SPLINE
SPL {X  -157.513, Y  +354.453, Z    +0.000, E1  +340.941, E3 -376360.122}
SPL {X  -159.408, Y  +368.861, Z    +0.000, E1  +348.865, E3 -376369.545}
SPL {X  -159.941, Y  +378.532, Z    +0.000, E1  +354.551, E3 -376373.150}
SPL {X  -159.990, Y  +383.966, Z    +0.000, E1  +358.149, E3 -376374.602}
SPL {X  -159.990, Y  +388.001, Z    +0.000, E1  +361.086, E3 -376375.537}
SPL {X  -159.990, Y  +392.647, Z    +0.000, E1  +364.974, E3 -376376.676}
SPL {X  -159.990, Y  +397.943, Z    +0.000, E1  +369.963, E3 -376378.260}
SPL {X  -159.990, Y  +406.530, Z    +0.000, E1  +377.917, E3 -376382.158}
SPL {X  -159.990, Y  +429.014, Z    +0.000, E1  +392.438, E3 -376400.815}
SPL {X  -159.990, Y  +437.635, Z    +0.000, E1  +395.495, E3 -376411.047}
SPL {X  -159.990, Y  +460.330, Z    +0.000, E1  +398.908, E3 -376451.734}
SPL {X  -159.990, Y  +464.953, Z    +0.000, E1  +398.907, E3 -376463.893}
SPL {X  -159.990, Y  +469.353, Z    +0.000, E1  +398.902, E3 -376475.473}
SPL {X  -159.990, Y  +475.034, Z    +0.000, E1  +398.936, E3 -376490.388}
SPL {X  -159.990, Y  +481.308, Z    +0.000, E1  +398.917, E3 -376506.899}
SPL {X  -159.990, Y  +486.996, Z    +0.000, E1  +398.928, E3 -376521.806}
SPL {X  -159.990, Y  +492.629, Z    +0.000, E1  +398.922, E3 -376536.613}
SPL {X  -159.990, Y  +497.431, Z    +0.000, E1  +398.905, E3 -376549.279}
SPL {X  -159.990, Y  +502.093, Z    +0.000, E1  +398.909, E3 -376561.554}
SPL {X  -159.990, Y  +507.821, Z    +0.000, E1  +398.930, E3 -376576.574}
SPL {X  -159.990, Y  +513.533, Z    +0.000, E1  +398.910, E3 -376591.633}
SPL {X  -159.990, Y  +518.435, Z    +0.000, E1  +398.905, E3 -376604.529}
SPL {X  -159.990, Y  +523.478, Z    +0.000, E1  +398.918, E3 -376617.757}
SPL {X  -159.990, Y  +528.627, Z    +0.000, E1  +398.910, E3 -376631.311}
SPL {X  -159.990, Y  +534.392, Z    +0.000, E1  +398.932, E3 -376646.441}
SPL {X  -159.990, Y  +540.299, Z    +0.000, E1  +398.912, E3 -376662.015}
SPL {X  -159.990, Y  +545.676, Z    +0.000, E1  +398.913, E3 -376676.153}
SPL {X  -159.990, Y  +550.777, Z    +0.000, E1  +398.906, E3 -376689.572}
SPL {X  -159.990, Y  +556.271, Z    +0.000, E1  +398.927, E3 -376703.975}
SPL {X  -159.990, Y  +561.696, Z    +0.000, E1  +398.912, E3 -376718.244}
SPL {X  -159.990, Y  +566.650, Z    +0.000, E1  +398.917, E3 -376731.258}
SPL {X  -159.990, Y  +571.814, Z    +0.000, E1  +398.914, E3 -376744.861}
SPL {X  -159.990, Y  +577.636, Z    +0.000, E1  +398.929, E3 -376760.158}
SPL {X  -159.990, Y  +583.167, Z    +0.000, E1  +398.906, E3 -376774.734}
SPL {X  -159.990, Y  +587.761, Z    +0.000, E1  +398.902, E3 -376786.819}
SPL {X  -159.990, Y  +592.962, Z    +0.000, E1  +398.925, E3 -376800.463}
SPL {X  -159.990, Y  +597.767, Z    +0.000, E1  +398.897, E3 -376813.138}
SPL {X  -159.990, Y  +602.727, Z    +0.000, E1  +398.920, E3 -376826.149}
SPL {X  -159.990, Y  +608.112, Z    +0.000, E1  +398.911, E3 -376840.323}
SPL {X  -159.990, Y  +613.039, Z    +0.000, E1  +398.906, E3 -376853.286}
SPL {X  -159.990, Y  +618.087, Z    +0.000, E1  +398.915, E3 -376866.544}
SPL {X  -159.990, Y  +623.264, Z    +0.000, E1  +398.906, E3 -376880.179}
SPL {X  -159.990, Y  +628.669, Z    +0.000, E1  +398.928, E3 -376894.347}
SPL {X  -159.990, Y  +634.089, Z    +0.000, E1  +398.907, E3 -376908.623}
SPL {X  -159.990, Y  +638.639, Z    +0.000, E1  +398.904, E3 -376920.608}
SPL {X  -159.990, Y  +643.555, Z    +0.000, E1  +398.910, E3 -376933.528}
SPL {X  -159.990, Y  +649.380, Z    +0.000, E1  +398.930, E3 -376948.806}
SPL {X  -159.990, Y  +654.813, Z    +0.000, E1  +398.905, E3 -376963.131}
SPL {X  -159.990, Y  +660.353, Z    +0.000, E1  +398.930, E3 -376977.662}
SPL {X  -159.990, Y  +665.703, Z    +0.000, E1  +398.903, E3 -376991.769}
SPL {X  -159.990, Y  +669.966, Z    +0.000, E1  +398.902, E3 -377002.976}
SPL {X  -159.954, Y  +674.895, Z    +0.000, E1  +398.910, E3 -377015.956}
SPL {X  -159.761, Y  +680.061, Z    +0.000, E1  +398.873, E3 -377029.735}
SPL {X  -159.443, Y  +684.716, Z    +0.000, E1  +398.815, E3 -377042.300}
SPL {X  -158.962, Y  +689.604, Z    +0.000, E1  +398.740, E3 -377055.669}
SPL {X  -158.318, Y  +694.567, Z    +0.000, E1  +398.614, E3 -377069.430}
SPL {X  -157.472, Y  +699.775, Z    +0.000, E1  +398.483, E3 -377083.990}
SPL {X  -156.506, Y  +704.705, Z    +0.000, E1  +398.294, E3 -377097.990}
SPL {X  -155.357, Y  +709.721, Z    +0.000, E1  +398.108, E3 -377112.345}
SPL {X  -154.005, Y  +714.851, Z    +0.000, E1  +397.854, E3 -377127.240}
SPL {X  -153.100, Y  +717.944, Z    +0.000, E1  +397.652, E3 -377136.350}
SPL {X  -151.080, Y  +724.146, Z    +0.000, E1  +393.201, E3 -377192.396}
ENDSPLINE

SPLINE
SPL {X  -157.921, Y  +697.149, Z    +0.000, E1  +377.701, E3 -377243.957}
SPL {X  -159.579, Y  +682.959, Z    +0.000, E1  +369.793, E3 -377251.905}
SPL {X  -159.938, Y  +675.561, Z    +0.000, E1  +365.399, E3 -377254.327}
SPL {X  -159.990, Y  +669.910, Z    +0.000, E1  +361.710, E3 -377255.618}
SPL {X  -159.990, Y  +665.465, Z    +0.000, E1  +358.378, E3 -377256.535}
SPL {X  -159.990, Y  +661.791, Z    +0.000, E1  +355.213, E3 -377257.373}
SPL {X  -159.990, Y  +656.991, Z    +0.000, E1  +350.742, E3 -377258.792}
SPL {X  -159.990, Y  +648.067, Z    +0.000, E1  +342.328, E3 -377262.522}
SPL {X  -159.990, Y  +620.451, Z    +0.000, E1  +325.419, E3 -377286.369}
SPL {X  -159.990, Y  +591.256, Z    +0.000, E1  +319.966, E3 -377332.863}
SPL {X  -159.990, Y  +586.740, Z    +0.000, E1  +319.956, E3 -377344.253}
SPL {X  -159.990, Y  +581.814, Z    +0.000, E1  +319.956, E3 -377356.692}
SPL {X  -159.990, Y  +577.274, Z    +0.000, E1  +319.964, E3 -377368.170}
SPL {X  -159.990, Y  +572.933, Z    +0.000, E1  +319.959, E3 -377379.111}
SPL {X  -159.990, Y  +568.504, Z    +0.000, E1  +319.956, E3 -377390.274}
SPL {X  -159.990, Y  +564.427, Z    +0.000, E1  +319.959, E3 -377400.560}
SPL {X  -159.990, Y  +558.823, Z    +0.000, E1  +319.916, E3 -377414.639}
SPL {X  -159.990, Y  +553.571, Z    +0.000, E1  +319.954, E3 -377427.921}
SPL {X  -159.990, Y  +549.413, Z    +0.000, E1  +319.938, E3 -377438.387}
SPL {X  -159.990, Y  +543.439, Z    +0.000, E1  +319.921, E3 -377453.475}
SPL {X  -159.990, Y  +537.213, Z    +0.000, E1  +319.937, E3 -377469.217}
SPL {X  -159.990, Y  +530.667, Z    +0.000, E1  +319.910, E3 -377485.675}
SPL {X  -159.990, Y  +523.984, Z    +0.000, E1  +319.922, E3 -377502.542}
SPL {X  -159.990, Y  +496.806, Z    +0.000, E1  +312.216, E3 -377516.457}
SPL {X  -159.990, Y  +490.245, Z    +0.000, E1  +312.831, E3 -377532.988}
SPL {X  -159.990, Y  +484.831, Z    +0.000, E1  +314.066, E3 -377551.220}
SPL {X  -159.990, Y  +480.580, Z    +0.000, E1  +315.242, E3 -377566.907}
SPL {X  -159.990, Y  +476.546, Z    +0.000, E1  +316.165, E3 -377581.202}
SPL {X  -159.990, Y  +472.671, Z    +0.000, E1  +317.192, E3 -377596.029}
SPL {X  -159.990, Y  +468.809, Z    +0.000, E1  +318.343, E3 -377611.957}
SPL {X  -159.990, Y  +465.057, Z    +0.000, E1  +319.375, E3 -377627.116}
SPL {X  -159.990, Y  +461.409, Z    +0.000, E1  +319.848, E3 -377639.015}
SPL {X  -159.990, Y  +456.934, Z    +0.000, E1  +319.854, E3 -377650.291}
SPL {X  -159.990, Y  +452.940, Z    +0.000, E1  +319.854, E3 -377660.336}
SPL {X  -159.990, Y  +448.856, Z    +0.000, E1  +319.859, E3 -377670.619}
SPL {X  -159.990, Y  +443.741, Z    +0.000, E1  +319.827, E3 -377683.437}
SPL {X  -159.990, Y  +436.703, Z    +0.000, E1  +319.809, E3 -377701.119}
SPL {X  -159.990, Y  +430.690, Z    +0.000, E1  +319.854, E3 -377716.312}
SPL {X  -159.990, Y  +426.145, Z    +0.000, E1  +319.853, E3 -377727.752}
SPL {X  -159.990, Y  +421.880, Z    +0.000, E1  +319.860, E3 -377738.485}
SPL {X  -159.990, Y  +417.572, Z    +0.000, E1  +319.852, E3 -377749.311}
SPL {X  -159.990, Y  +412.619, Z    +0.000, E1  +319.850, E3 -377761.803}
SPL {X  -159.990, Y  +406.264, Z    +0.000, E1  +319.825, E3 -377777.751}
SPL {X  -159.990, Y  +400.535, Z    +0.000, E1  +319.859, E3 -377792.214}
SPL {X  -159.990, Y  +396.024, Z    +0.000, E1  +319.860, E3 -377803.570}
SPL {X  -159.990, Y  +391.614, Z    +0.000, E1  +319.860, E3 -377814.663}
SPL {X  -159.990, Y  +387.212, Z    +0.000, E1  +319.859, E3 -377825.736}
SPL {X  -159.990, Y  +382.743, Z    +0.000, E1  +319.857, E3 -377836.977}
SPL {X  -159.925, Y  +377.946, Z    +0.000, E1  +319.864, E3 -377849.114}
SPL {X  -159.703, Y  +372.915, Z    +0.000, E1  +319.904, E3 -377862.014}
SPL {X  -159.358, Y  +368.290, Z    +0.000, E1  +319.961, E3 -377873.976}
SPL {X  -158.955, Y  +364.333, Z    +0.000, E1  +320.046, E3 -377884.379}
SPL {X  -158.482, Y  +360.589, Z    +0.000, E1  +320.125, E3 -377894.305}
SPL {X  -157.729, Y  +355.695, Z    +0.000, E1  +320.237, E3 -377907.378}
SPL {X  -156.893, Y  +351.173, Z    +0.000, E1  +320.410, E3 -377919.661}
SPL {X  -156.148, Y  +347.650, Z    +0.000, E1  +320.549, E3 -377929.307}
SPL {X  -155.268, Y  +343.918, Z    +0.000, E1  +320.696, E3 -377939.588}
SPL {X  -153.936, Y  +338.906, Z    +0.000, E1  +320.911, E3 -377953.527}
SPL {X  -152.628, Y  +334.526, Z    +0.000, E1  +321.188, E3 -377965.929}
SPL {X  -151.010, Y  +329.654, Z    +0.000, E1  +326.674, E3 -378023.765}
ENDSPLINE

SPLINE
SPL {X  -157.513, Y  +354.453, Z    +0.000, E1  +340.941, E3 -378069.799}
SPL {X  -159.408, Y  +368.861, Z    +0.000, E1  +348.865, E3 -378079.222}
SPL {X  -159.941, Y  +378.532, Z    +0.000, E1  +354.551, E3 -378082.828}
SPL {X  -159.990, Y  +383.966, Z    +0.000, E1  +358.149, E3 -378084.280}
SPL {X  -159.990, Y  +388.001, Z    +0.000, E1  +361.086, E3 -378085.215}
SPL {X  -159.990, Y  +392.647, Z    +0.000, E1  +364.974, E3 -378086.353}
SPL {X  -159.990, Y  +397.943, Z    +0.000, E1  +369.963, E3 -378087.938}
SPL {X  -159.990, Y  +407.689, Z    +0.000, E1  +378.860, E3 -378092.592}
SPL {X  -159.990, Y  +434.822, Z    +0.000, E1  +394.625, E3 -378117.136}
SPL {X  -159.990, Y  +460.330, Z    +0.000, E1  +398.908, E3 -378161.412}
SPL {X  -159.990, Y  +464.953, Z    +0.000, E1  +398.907, E3 -378173.570}
SPL {X  -159.990, Y  +469.353, Z    +0.000, E1  +398.902, E3 -378185.150}
SPL {X  -159.990, Y  +475.034, Z    +0.000, E1  +398.936, E3 -378200.065}
SPL {X  -159.990, Y  +481.308, Z    +0.000, E1  +398.917, E3 -378216.576}
SPL {X  -159.990, Y  +485.396, Z    +0.000, E1  +398.893, E3 -378227.336}
SPL {X  -159.990, Y  +489.893, Z    +0.000, E1  +398.930, E3 -378239.091}
SPL {X  -159.990, Y  +496.271, Z    +0.000, E1  +398.942, E3 -378255.847}
SPL {X  -159.990, Y  +502.093, Z    +0.000, E1  +398.909, E3 -378271.231}
SPL {X  -159.990, Y  +507.821, Z    +0.000, E1  +398.930, E3 -378286.251}
SPL {X  -159.990, Y  +513.533, Z    +0.000, E1  +398.910, E3 -378301.311}
SPL {X  -159.990, Y  +518.435, Z    +0.000, E1  +398.905, E3 -378314.206}
SPL {X  -159.990, Y  +523.478, Z    +0.000, E1  +398.918, E3 -378327.435}
SPL {X  -159.990, Y  +528.627, Z    +0.000, E1  +398.910, E3 -378340.988}
SPL {X  -159.990, Y  +533.053, Z    +0.000, E1  +398.899, E3 -378352.646}
SPL {X  -159.990, Y  +537.174, Z    +0.000, E1  +398.910, E3 -378363.460}
SPL {X  -159.990, Y  +541.259, Z    +0.000, E1  +398.888, E3 -378374.260}
SPL {X  -159.990, Y  +545.676, Z    +0.000, E1  +398.913, E3 -378385.831}
SPL {X  -159.990, Y  +550.777, Z    +0.000, E1  +398.906, E3 -378399.250}
SPL {X  -159.990, Y  +554.638, Z    +0.000, E1  +398.890, E3 -378409.420}
SPL {X  -159.990, Y  +557.678, Z    +0.000, E1  +398.893, E3 -378417.396}
SPL {X  -159.990, Y  +561.696, Z    +0.000, E1  +398.912, E3 -378427.922}
SPL {X  -159.990, Y  +566.650, Z    +0.000, E1  +398.917, E3 -378440.935}
SPL {X  -159.990, Y  +571.814, Z    +0.000, E1  +398.914, E3 -378454.538}
SPL {X  -159.990, Y  +576.364, Z    +0.000, E1  +398.896, E3 -378466.541}
SPL {X  -159.990, Y  +582.060, Z    +0.000, E1  +398.942, E3 -378481.447}
SPL {X  -159.990, Y  +589.106, Z    +0.000, E1  +398.939, E3 -378499.978}
SPL {X  -159.990, Y  +596.185, Z    +0.000, E1  +398.945, E3 -378518.587}
SPL {X  -159.990, Y  +602.727, Z    +0.000, E1  +398.920, E3 -378535.826}
SPL {X  -159.990, Y  +608.112, Z    +0.000, E1  +398.911, E3 -378550.001}
SPL {X  -159.990, Y  +614.125, Z    +0.000, E1  +398.936, E3 -378565.776}
SPL {X  -159.990, Y  +619.061, Z    +0.000, E1  +398.894, E3 -378578.807}
SPL {X  -159.990, Y  +623.264, Z    +0.000, E1  +398.906, E3 -378589.856}
SPL {X  -159.990, Y  +628.669, Z    +0.000, E1  +398.928, E3 -378604.025}
SPL {X  -159.990, Y  +634.089, Z    +0.000, E1  +398.907, E3 -378618.300}
SPL {X  -159.990, Y  +638.639, Z    +0.000, E1  +398.904, E3 -378630.286}
SPL {X  -159.990, Y  +644.750, Z    +0.000, E1  +398.946, E3 -378646.291}
SPL {X  -159.990, Y  +650.458, Z    +0.000, E1  +398.900, E3 -378661.364}
SPL {X  -159.990, Y  +654.813, Z    +0.000, E1  +398.905, E3 -378672.808}
SPL {X  -159.990, Y  +660.353, Z    +0.000, E1  +398.930, E3 -378687.339}
SPL {X  -159.990, Y  +665.703, Z    +0.000, E1  +398.903, E3 -378701.447}
SPL {X  -159.990, Y  +669.966, Z    +0.000, E1  +398.902, E3 -378712.653}
SPL {X  -159.954, Y  +674.895, Z    +0.000, E1  +398.910, E3 -378725.633}
SPL {X  -159.761, Y  +680.061, Z    +0.000, E1  +398.873, E3 -378739.412}
SPL {X  -159.443, Y  +684.716, Z    +0.000, E1  +398.815, E3 -378751.977}
SPL {X  -158.962, Y  +689.604, Z    +0.000, E1  +398.740, E3 -378765.346}
SPL {X  -158.139, Y  +695.766, Z    +0.000, E1  +398.623, E3 -378782.392}
SPL {X  -157.275, Y  +700.848, Z    +0.000, E1  +398.415, E3 -378796.744}
SPL {X  -156.506, Y  +704.705, Z    +0.000, E1  +398.294, E3 -378807.668}
SPL {X  -155.357, Y  +709.721, Z    +0.000, E1  +398.108, E3 -378822.023}
SPL {X  -154.286, Y  +713.838, Z    +0.000, E1  +397.877, E3 -378834.005}
SPL {X  -153.345, Y  +717.131, Z    +0.000, E1  +397.713, E3 -378843.619}
SPL {X  -151.080, Y  +724.146, Z    +0.000, E1  +393.201, E3 -378902.073}
ENDSPLINE

SPLINE
SPL {X  -157.921, Y  +697.149, Z    +0.000, E1  +377.701, E3 -378953.634}
SPL {X  -159.579, Y  +682.959, Z    +0.000, E1  +369.793, E3 -378961.582}
SPL {X  -159.938, Y  +675.561, Z    +0.000, E1  +365.399, E3 -378964.005}
SPL {X  -159.990, Y  +669.910, Z    +0.000, E1  +361.710, E3 -378965.295}
SPL {X  -159.990, Y  +665.465, Z    +0.000, E1  +358.378, E3 -378966.213}
SPL {X  -159.990, Y  +661.791, Z    +0.000, E1  +355.213, E3 -378967.051}
SPL {X  -159.990, Y  +656.991, Z    +0.000, E1  +350.742, E3 -378968.470}
SPL {X  -159.990, Y  +648.067, Z    +0.000, E1  +342.328, E3 -378972.199}
SPL {X  -159.990, Y  +620.451, Z    +0.000, E1  +325.419, E3 -378996.047}
SPL {X  -159.990, Y  +591.256, Z    +0.000, E1  +319.966, E3 -379042.540}
SPL {X  -159.990, Y  +586.740, Z    +0.000, E1  +319.956, E3 -379053.930}
SPL {X  -159.990, Y  +581.814, Z    +0.000, E1  +319.956, E3 -379066.370}
SPL {X  -159.990, Y  +577.274, Z    +0.000, E1  +319.964, E3 -379077.847}
SPL {X  -159.990, Y  +572.933, Z    +0.000, E1  +319.959, E3 -379088.789}
SPL {X  -159.990, Y  +568.504, Z    +0.000, E1  +319.956, E3 -379099.951}
SPL {X  -159.990, Y  +563.189, Z    +0.000, E1  +319.932, E3 -379113.325}
SPL {X  -159.990, Y  +557.707, Z    +0.000, E1  +319.949, E3 -379127.180}
SPL {X  -159.990, Y  +552.104, Z    +0.000, E1  +319.922, E3 -379141.255}
SPL {X  -159.990, Y  +545.912, Z    +0.000, E1  +319.929, E3 -379156.904}
SPL {X  -159.990, Y  +540.054, Z    +0.000, E1  +319.939, E3 -379171.732}
SPL {X  -159.990, Y  +535.835, Z    +0.000, E1  +319.966, E3 -379182.412}
SPL {X  -159.990, Y  +530.667, Z    +0.000, E1  +319.910, E3 -379195.353}
SPL {X  -159.990, Y  +523.984, Z    +0.000, E1  +319.922, E3 -379212.219}
SPL {X  -159.990, Y  +496.806, Z    +0.000, E1  +312.216, E3 -379226.134}
SPL {X  -159.990, Y  +490.245, Z    +0.000, E1  +312.831, E3 -379242.665}
SPL {X  -159.990, Y  +486.737, Z    +0.000, E1  +313.729, E3 -379254.671}
SPL {X  -159.990, Y  +483.955, Z    +0.000, E1  +314.316, E3 -379263.963}
SPL {X  -159.990, Y  +480.580, Z    +0.000, E1  +315.242, E3 -379276.584}
SPL {X  -159.990, Y  +476.546, Z    +0.000, E1  +316.165, E3 -379290.879}
SPL {X  -159.990, Y  +473.377, Z    +0.000, E1  +316.953, E3 -379302.493}
SPL {X  -159.990, Y  +470.788, Z    +0.000, E1  +317.853, E3 -379313.907}
SPL {X  -159.990, Y  +467.944, Z    +0.000, E1  +318.635, E3 -379325.228}
SPL {X  -159.990, Y  +465.057, Z    +0.000, E1  +319.375, E3 -379336.793}
SPL {X  -159.990, Y  +461.409, Z    +0.000, E1  +319.848, E3 -379348.693}
SPL {X  -159.990, Y  +456.934, Z    +0.000, E1  +319.854, E3 -379359.968}
SPL {X  -159.990, Y  +452.940, Z    +0.000, E1  +319.854, E3 -379370.013}
SPL {X  -159.990, Y  +448.856, Z    +0.000, E1  +319.859, E3 -379380.296}
SPL {X  -159.990, Y  +444.973, Z    +0.000, E1  +319.856, E3 -379390.062}
SPL {X  -159.990, Y  +439.927, Z    +0.000, E1  +319.837, E3 -379402.718}
SPL {X  -159.990, Y  +435.246, Z    +0.000, E1  +319.853, E3 -379414.527}
SPL {X  -159.990, Y  +430.690, Z    +0.000, E1  +319.854, E3 -379425.989}
SPL {X  -159.990, Y  +426.145, Z    +0.000, E1  +319.853, E3 -379437.429}
SPL {X  -159.990, Y  +421.880, Z    +0.000, E1  +319.860, E3 -379448.162}
SPL {X  -159.990, Y  +416.246, Z    +0.000, E1  +319.819, E3 -379462.291}
SPL {X  -159.990, Y  +409.936, Z    +0.000, E1  +319.849, E3 -379478.227}
SPL {X  -159.990, Y  +404.988, Z    +0.000, E1  +319.861, E3 -379490.693}
SPL {X  -159.990, Y  +400.535, Z    +0.000, E1  +319.859, E3 -379501.891}
SPL {X  -159.990, Y  +396.024, Z    +0.000, E1  +319.860, E3 -379513.247}
SPL {X  -159.990, Y  +391.614, Z    +0.000, E1  +319.860, E3 -379524.341}
SPL {X  -159.990, Y  +387.212, Z    +0.000, E1  +319.859, E3 -379535.413}
SPL {X  -159.990, Y  +382.743, Z    +0.000, E1  +319.857, E3 -379546.655}
SPL {X  -159.925, Y  +377.946, Z    +0.000, E1  +319.864, E3 -379558.791}
SPL {X  -159.703, Y  +372.915, Z    +0.000, E1  +319.904, E3 -379571.691}
SPL {X  -159.358, Y  +368.290, Z    +0.000, E1  +319.961, E3 -379583.654}
SPL {X  -158.955, Y  +364.333, Z    +0.000, E1  +320.046, E3 -379594.056}
SPL {X  -158.270, Y  +359.106, Z    +0.000, E1  +320.118, E3 -379607.867}
SPL {X  -157.143, Y  +352.453, Z    +0.000, E1  +320.322, E3 -379625.798}
SPL {X  -156.148, Y  +347.650, Z    +0.000, E1  +320.549, E3 -379638.984}
SPL {X  -155.268, Y  +343.918, Z    +0.000, E1  +320.696, E3 -379649.265}
SPL {X  -154.153, Y  +339.677, Z    +0.000, E1  +320.896, E3 -379661.072}
SPL {X  -152.885, Y  +335.352, Z    +0.000, E1  +321.114, E3 -379673.226}
SPL {X  -151.010, Y  +329.654, Z    +0.000, E1  +326.674, E3 -379733.442}
ENDSPLINE

SPLINE
SPL {X  -157.513, Y  +354.453, Z    +0.000, E1  +340.941, E3 -379779.477}
SPL {X  -159.408, Y  +368.861, Z    +0.000, E1  +348.865, E3 -379788.899}
SPL {X  -159.941, Y  +378.532, Z    +0.000, E1  +354.551, E3 -379792.505}
SPL {X  -159.990, Y  +383.966, Z    +0.000, E1  +358.149, E3 -379793.957}
SPL {X  -159.990, Y  +389.165, Z    +0.000, E1  +361.929, E3 -379795.159}
SPL {X  -159.990, Y  +394.164, Z    +0.000, E1  +366.430, E3 -379796.451}
SPL {X  -159.990, Y  +399.434, Z    +0.000, E1  +371.306, E3 -379798.211}
SPL {X  -159.990, Y  +407.956, Z    +0.000, E1  +379.215, E3 -379802.299}
SPL {X  -159.990, Y  +429.014, Z    +0.000, E1  +392.438, E3 -379820.170}
SPL {X  -159.990, Y  +437.635, Z    +0.000, E1  +395.495, E3 -379830.402}
SPL {X  -159.990, Y  +460.330, Z    +0.000, E1  +398.908, E3 -379871.089}
SPL {X  -159.990, Y  +464.953, Z    +0.000, E1  +398.907, E3 -379883.247}
SPL {X  -159.990, Y  +469.353, Z    +0.000, E1  +398.902, E3 -379894.828}
SPL {X  -159.990, Y  +473.222, Z    +0.000, E1  +398.891, E3 -379905.036}
SPL {X  -159.990, Y  +477.957, Z    +0.000, E1  +398.922, E3 -379917.442}
SPL {X  -159.990, Y  +482.463, Z    +0.000, E1  +398.891, E3 -379929.329}
SPL {X  -159.990, Y  +486.996, Z    +0.000, E1  +398.928, E3 -379941.161}
SPL {X  -159.990, Y  +492.629, Z    +0.000, E1  +398.922, E3 -379955.968}
SPL {X  -159.990, Y  +497.431, Z    +0.000, E1  +398.905, E3 -379968.634}
SPL {X  -159.990, Y  +502.093, Z    +0.000, E1  +398.909, E3 -379980.909}
SPL {X  -159.990, Y  +507.821, Z    +0.000, E1  +398.930, E3 -379995.929}
SPL {X  -159.990, Y  +513.533, Z    +0.000, E1  +398.910, E3 -380010.988}
SPL {X  -159.990, Y  +518.435, Z    +0.000, E1  +398.905, E3 -380023.883}
SPL {X  -159.990, Y  +523.478, Z    +0.000, E1  +398.918, E3 -380037.112}
SPL {X  -159.990, Y  +528.627, Z    +0.000, E1  +398.910, E3 -380050.666}
SPL {X  -159.990, Y  +533.053, Z    +0.000, E1  +398.899, E3 -380062.323}
SPL {X  -159.990, Y  +537.174, Z    +0.000, E1  +398.910, E3 -380073.138}
SPL {X  -159.990, Y  +541.259, Z    +0.000, E1  +398.888, E3 -380083.937}
SPL {X  -159.990, Y  +545.676, Z    +0.000, E1  +398.913, E3 -380095.508}
SPL {X  -159.990, Y  +550.777, Z    +0.000, E1  +398.906, E3 -380108.927}
SPL {X  -159.990, Y  +556.271, Z    +0.000, E1  +398.927, E3 -380123.330}
SPL {X  -159.990, Y  +561.696, Z    +0.000, E1  +398.912, E3 -380137.599}
SPL {X  -159.990, Y  +566.650, Z    +0.000, E1  +398.917, E3 -380150.613}
SPL {X  -159.990, Y  +571.814, Z    +0.000, E1  +398.914, E3 -380164.216}
SPL {X  -159.990, Y  +576.364, Z    +0.000, E1  +398.896, E3 -380176.219}
SPL {X  -159.990, Y  +582.060, Z    +0.000, E1  +398.942, E3 -380191.124}
SPL {X  -159.990, Y  +587.761, Z    +0.000, E1  +398.902, E3 -380206.173}
SPL {X  -159.990, Y  +592.962, Z    +0.000, E1  +398.925, E3 -380219.817}
SPL {X  -159.990, Y  +599.478, Z    +0.000, E1  +398.941, E3 -380236.928}
SPL {X  -159.990, Y  +606.904, Z    +0.000, E1  +398.953, E3 -380256.441}
SPL {X  -159.990, Y  +613.039, Z    +0.000, E1  +398.906, E3 -380272.641}
SPL {X  -159.990, Y  +618.087, Z    +0.000, E1  +398.915, E3 -380285.899}
SPL {X  -159.990, Y  +623.264, Z    +0.000, E1  +398.906, E3 -380299.534}
SPL {X  -159.990, Y  +628.669, Z    +0.000, E1  +398.928, E3 -380313.702}
SPL {X  -159.990, Y  +634.089, Z    +0.000, E1  +398.907, E3 -380327.978}
SPL {X  -159.990, Y  +638.639, Z    +0.000, E1  +398.904, E3 -380339.963}
SPL {X  -159.990, Y  +644.750, Z    +0.000, E1  +398.946, E3 -380355.969}
SPL {X  -159.990, Y  +650.458, Z    +0.000, E1  +398.900, E3 -380371.041}
SPL {X  -159.990, Y  +654.813, Z    +0.000, E1  +398.905, E3 -380382.485}
SPL {X  -159.990, Y  +660.353, Z    +0.000, E1  +398.930, E3 -380397.017}
SPL {X  -159.990, Y  +665.703, Z    +0.000, E1  +398.903, E3 -380411.124}
SPL {X  -159.990, Y  +671.472, Z    +0.000, E1  +398.942, E3 -380426.229}
SPL {X  -159.920, Y  +676.216, Z    +0.000, E1  +398.875, E3 -380438.864}
SPL {X  -159.761, Y  +680.061, Z    +0.000, E1  +398.873, E3 -380449.089}
SPL {X  -159.327, Y  +686.045, Z    +0.000, E1  +398.835, E3 -380465.212}
SPL {X  -158.832, Y  +690.714, Z    +0.000, E1  +398.685, E3 -380478.138}
SPL {X  -158.318, Y  +694.567, Z    +0.000, E1  +398.614, E3 -380488.785}
SPL {X  -157.472, Y  +699.775, Z    +0.000, E1  +398.483, E3 -380503.345}
SPL {X  -156.506, Y  +704.705, Z    +0.000, E1  +398.294, E3 -380517.345}
SPL {X  -155.680, Y  +708.387, Z    +0.000, E1  +398.127, E3 -380527.916}
SPL {X  -154.586, Y  +712.730, Z    +0.000, E1  +397.967, E3 -380540.413}
SPL {X  -153.345, Y  +717.131, Z    +0.000, E1  +397.713, E3 -380553.297}
SPL {X  -151.080, Y  +724.146, Z    +0.000, E1  +393.201, E3 -380611.751}
ENDSPLINE

SPLINE
SPL {X  -157.921, Y  +697.149, Z    +0.000, E1  +377.701, E3 -380663.311}
SPL {X  -159.579, Y  +682.959, Z    +0.000, E1  +369.793, E3 -380671.260}
SPL {X  -159.938, Y  +675.561, Z    +0.000, E1  +365.399, E3 -380673.682}
SPL {X  -159.990, Y  +669.910, Z    +0.000, E1  +361.710, E3 -380674.973}
SPL {X  -159.990, Y  +665.465, Z    +0.000, E1  +358.378, E3 -380675.890}
SPL {X  -159.990, Y  +661.791, Z    +0.000, E1  +355.213, E3 -380676.728}
SPL {X  -159.990, Y  +656.991, Z    +0.000, E1  +350.742, E3 -380678.147}
SPL {X  -159.990, Y  +648.067, Z    +0.000, E1  +342.328, E3 -380681.877}
SPL {X  -159.990, Y  +620.451, Z    +0.000, E1  +325.419, E3 -380705.724}
SPL {X  -159.990, Y  +591.256, Z    +0.000, E1  +319.966, E3 -380752.217}
SPL {X  -159.990, Y  +586.740, Z    +0.000, E1  +319.956, E3 -380763.608}
SPL {X  -159.990, Y  +581.814, Z    +0.000, E1  +319.956, E3 -380776.047}
SPL {X  -159.990, Y  +577.274, Z    +0.000, E1  +319.964, E3 -380787.525}
SPL {X  -159.990, Y  +572.933, Z    +0.000, E1  +319.959, E3 -380798.466}
SPL {X  -159.990, Y  +568.504, Z    +0.000, E1  +319.956, E3 -380809.629}
SPL {X  -159.990, Y  +563.189, Z    +0.000, E1  +319.932, E3 -380823.002}
SPL {X  -159.990, Y  +557.707, Z    +0.000, E1  +319.949, E3 -380836.857}
SPL {X  -159.990, Y  +553.571, Z    +0.000, E1  +319.954, E3 -380847.276}
SPL {X  -159.990, Y  +549.413, Z    +0.000, E1  +319.938, E3 -380857.742}
SPL {X  -159.990, Y  +544.924, Z    +0.000, E1  +319.955, E3 -380869.123}
SPL {X  -159.990, Y  +540.054, Z    +0.000, E1  +319.939, E3 -380881.409}
SPL {X  -159.990, Y  +533.683, Z    +0.000, E1  +319.916, E3 -380897.434}
SPL {X  -159.990, Y  +528.899, Z    +0.000, E1  +319.955, E3 -380909.550}
SPL {X  -159.990, Y  +523.984, Z    +0.000, E1  +319.922, E3 -380921.897}
SPL {X  -159.990, Y  +502.378, Z    +0.000, E1  +313.079, E3 -380930.008}
SPL {X  -159.990, Y  +493.568, Z    +0.000, E1  +312.053, E3 -380941.175}
SPL {X  -159.990, Y  +489.464, Z    +0.000, E1  +313.059, E3 -380955.042}
SPL {X  -159.990, Y  +484.831, Z    +0.000, E1  +314.066, E3 -380970.575}
SPL {X  -159.990, Y  +480.580, Z    +0.000, E1  +315.242, E3 -380986.262}
SPL {X  -159.990, Y  +476.546, Z    +0.000, E1  +316.165, E3 -381000.556}
SPL {X  -159.990, Y  +472.671, Z    +0.000, E1  +317.192, E3 -381015.384}
SPL {X  -159.990, Y  +468.809, Z    +0.000, E1  +318.343, E3 -381031.312}
SPL {X  -159.990, Y  +465.057, Z    +0.000, E1  +319.375, E3 -381046.471}
SPL {X  -159.990, Y  +461.409, Z    +0.000, E1  +319.848, E3 -381058.370}
SPL {X  -159.990, Y  +456.934, Z    +0.000, E1  +319.854, E3 -381069.646}
SPL {X  -159.990, Y  +452.940, Z    +0.000, E1  +319.854, E3 -381079.691}
SPL {X  -159.990, Y  +448.856, Z    +0.000, E1  +319.859, E3 -381089.974}
SPL {X  -159.990, Y  +443.741, Z    +0.000, E1  +319.827, E3 -381102.792}
SPL {X  -159.990, Y  +436.703, Z    +0.000, E1  +319.809, E3 -381120.474}
SPL {X  -159.990, Y  +430.690, Z    +0.000, E1  +319.854, E3 -381135.667}
SPL {X  -159.990, Y  +426.145, Z    +0.000, E1  +319.853, E3 -381147.106}
SPL {X  -159.990, Y  +421.880, Z    +0.000, E1  +319.860, E3 -381157.839}
SPL {X  -159.990, Y  +417.572, Z    +0.000, E1  +319.852, E3 -381168.666}
SPL {X  -159.990, Y  +412.619, Z    +0.000, E1  +319.850, E3 -381181.158}
SPL {X  -159.990, Y  +406.264, Z    +0.000, E1  +319.825, E3 -381197.106}
SPL {X  -159.990, Y  +400.535, Z    +0.000, E1  +319.859, E3 -381211.569}
SPL {X  -159.990, Y  +396.024, Z    +0.000, E1  +319.860, E3 -381222.925}
SPL {X  -159.990, Y  +391.614, Z    +0.000, E1  +319.860, E3 -381234.018}
SPL {X  -159.990, Y  +387.212, Z    +0.000, E1  +319.859, E3 -381245.090}
SPL {X  -159.990, Y  +382.743, Z    +0.000, E1  +319.857, E3 -381256.332}
SPL {X  -159.925, Y  +377.946, Z    +0.000, E1  +319.864, E3 -381268.469}
SPL {X  -159.703, Y  +372.915, Z    +0.000, E1  +319.904, E3 -381281.369}
SPL {X  -159.358, Y  +368.290, Z    +0.000, E1  +319.961, E3 -381293.331}
SPL {X  -158.955, Y  +364.333, Z    +0.000, E1  +320.046, E3 -381303.734}
SPL {X  -158.482, Y  +360.589, Z    +0.000, E1  +320.125, E3 -381313.660}
SPL {X  -157.729, Y  +355.695, Z    +0.000, E1  +320.237, E3 -381326.733}
SPL {X  -156.893, Y  +351.173, Z    +0.000, E1  +320.410, E3 -381339.016}
SPL {X  -156.148, Y  +347.650, Z    +0.000, E1  +320.549, E3 -381348.662}
SPL {X  -155.268, Y  +343.918, Z    +0.000, E1  +320.696, E3 -381358.943}
SPL {X  -154.153, Y  +339.677, Z    +0.000, E1  +320.896, E3 -381370.749}
SPL {X  -152.885, Y  +335.352, Z    +0.000, E1  +321.114, E3 -381382.904}
SPL {X  -151.010, Y  +329.654, Z    +0.000, E1  +326.674, E3 -381443.120}
ENDSPLINE

SPLINE
SPL {X  -157.513, Y  +354.453, Z    +0.000, E1  +340.941, E3 -381489.154}
SPL {X  -159.408, Y  +368.861, Z    +0.000, E1  +348.865, E3 -381498.577}
SPL {X  -159.941, Y  +378.532, Z    +0.000, E1  +354.551, E3 -381502.182}
SPL {X  -159.990, Y  +383.966, Z    +0.000, E1  +358.149, E3 -381503.634}
SPL {X  -159.990, Y  +389.165, Z    +0.000, E1  +361.929, E3 -381504.836}
SPL {X  -159.990, Y  +394.164, Z    +0.000, E1  +366.430, E3 -381506.129}
SPL {X  -159.990, Y  +399.434, Z    +0.000, E1  +371.306, E3 -381507.888}
SPL {X  -159.990, Y  +407.956, Z    +0.000, E1  +379.215, E3 -381511.977}
SPL {X  -159.990, Y  +429.014, Z    +0.000, E1  +392.438, E3 -381529.847}
SPL {X  -159.990, Y  +437.635, Z    +0.000, E1  +395.495, E3 -381540.079}
SPL {X  -159.990, Y  +460.330, Z    +0.000, E1  +398.908, E3 -381580.767}
SPL {X  -159.990, Y  +464.953, Z    +0.000, E1  +398.907, E3 -381592.925}
SPL {X  -159.990, Y  +469.353, Z    +0.000, E1  +398.902, E3 -381604.505}
SPL {X  -159.990, Y  +475.034, Z    +0.000, E1  +398.936, E3 -381619.420}
SPL {X  -159.990, Y  +481.308, Z    +0.000, E1  +398.917, E3 -381635.931}
SPL {X  -159.990, Y  +486.996, Z    +0.000, E1  +398.928, E3 -381650.839}
SPL {X  -159.990, Y  +492.629, Z    +0.000, E1  +398.922, E3 -381665.645}
SPL {X  -159.990, Y  +497.431, Z    +0.000, E1  +398.905, E3 -381678.312}
SPL {X  -159.990, Y  +502.093, Z    +0.000, E1  +398.909, E3 -381690.586}
SPL {X  -159.990, Y  +507.821, Z    +0.000, E1  +398.930, E3 -381705.606}
SPL {X  -159.990, Y  +513.533, Z    +0.000, E1  +398.910, E3 -381720.666}
SPL {X  -159.990, Y  +519.462, Z    +0.000, E1  +398.933, E3 -381736.218}
SPL {X  -159.990, Y  +524.415, Z    +0.000, E1  +398.896, E3 -381749.283}
SPL {X  -159.990, Y  +528.627, Z    +0.000, E1  +398.910, E3 -381760.343}
SPL {X  -159.990, Y  +533.053, Z    +0.000, E1  +398.899, E3 -381772.001}
SPL {X  -159.990, Y  +537.174, Z    +0.000, E1  +398.910, E3 -381782.815}
SPL {X  -159.990, Y  +541.259, Z    +0.000, E1  +398.888, E3 -381793.615}
SPL {X  -159.990, Y  +545.676, Z    +0.000, E1  +398.913, E3 -381805.185}
SPL {X  -159.990, Y  +550.777, Z    +0.000, E1  +398.906, E3 -381818.605}
SPL {X  -159.990, Y  +556.271, Z    +0.000, E1  +398.927, E3 -381833.007}
SPL {X  -159.990, Y  +561.696, Z    +0.000, E1  +398.912, E3 -381847.277}
SPL {X  -159.990, Y  +566.650, Z    +0.000, E1  +398.917, E3 -381860.290}
SPL {X  -159.990, Y  +571.814, Z    +0.000, E1  +398.914, E3 -381873.893}
SPL {X  -159.990, Y  +577.636, Z    +0.000, E1  +398.929, E3 -381889.190}
SPL {X  -159.990, Y  +583.167, Z    +0.000, E1  +398.906, E3 -381903.766}
SPL {X  -159.990, Y  +589.106, Z    +0.000, E1  +398.939, E3 -381919.333}
SPL {X  -159.990, Y  +596.185, Z    +0.000, E1  +398.945, E3 -381937.942}
SPL {X  -159.990, Y  +602.727, Z    +0.000, E1  +398.920, E3 -381955.181}
SPL {X  -159.990, Y  +608.112, Z    +0.000, E1  +398.911, E3 -381969.355}
SPL {X  -159.990, Y  +614.125, Z    +0.000, E1  +398.936, E3 -381985.131}
SPL {X  -159.990, Y  +619.061, Z    +0.000, E1  +398.894, E3 -381998.162}
SPL {X  -159.990, Y  +623.264, Z    +0.000, E1  +398.906, E3 -382009.211}
SPL {X  -159.990, Y  +628.669, Z    +0.000, E1  +398.928, E3 -382023.379}
SPL {X  -159.990, Y  +634.089, Z    +0.000, E1  +398.907, E3 -382037.655}
SPL {X  -159.990, Y  +638.639, Z    +0.000, E1  +398.904, E3 -382049.641}
SPL {X  -159.990, Y  +644.750, Z    +0.000, E1  +398.946, E3 -382065.646}
SPL {X  -159.990, Y  +650.458, Z    +0.000, E1  +398.900, E3 -382080.719}
SPL {X  -159.990, Y  +654.813, Z    +0.000, E1  +398.905, E3 -382092.163}
SPL {X  -159.990, Y  +658.715, Z    +0.000, E1  +398.892, E3 -382102.444}
SPL {X  -159.990, Y  +661.848, Z    +0.000, E1  +398.892, E3 -382110.682}
SPL {X  -159.990, Y  +665.703, Z    +0.000, E1  +398.903, E3 -382120.801}
SPL {X  -159.990, Y  +669.966, Z    +0.000, E1  +398.902, E3 -382132.008}
SPL {X  -159.954, Y  +674.895, Z    +0.000, E1  +398.910, E3 -382144.988}
SPL {X  -159.761, Y  +680.061, Z    +0.000, E1  +398.873, E3 -382158.767}
SPL {X  -159.443, Y  +684.716, Z    +0.000, E1  +398.815, E3 -382171.332}
SPL {X  -158.962, Y  +689.604, Z    +0.000, E1  +398.740, E3 -382184.701}
SPL {X  -158.318, Y  +694.567, Z    +0.000, E1  +398.614, E3 -382198.462}
SPL {X  -157.472, Y  +699.775, Z    +0.000, E1  +398.483, E3 -382213.022}
SPL {X  -156.506, Y  +704.705, Z    +0.000, E1  +398.294, E3 -382227.022}
SPL {X  -155.357, Y  +709.721, Z    +0.000, E1  +398.108, E3 -382241.377}
SPL {X  -154.286, Y  +713.838, Z    +0.000, E1  +397.877, E3 -382253.360}
SPL {X  -153.345, Y  +717.131, Z    +0.000, E1  +397.713, E3 -382262.974}
SPL {X  -151.080, Y  +724.146, Z    +0.000, E1  +393.201, E3 -382321.428}
ENDSPLINE

SPLINE
SPL {X  -157.921, Y  +697.149, Z    +0.000, E1  +377.701, E3 -382372.989}
SPL {X  -159.579, Y  +682.959, Z    +0.000, E1  +369.793, E3 -382380.937}
SPL {X  -159.938, Y  +675.561, Z    +0.000, E1  +365.399, E3 -382383.359}
SPL {X  -159.990, Y  +669.910, Z    +0.000, E1  +361.710, E3 -382384.650}
SPL {X  -159.990, Y  +665.465, Z    +0.000, E1  +358.378, E3 -382385.568}
SPL {X  -159.990, Y  +661.791, Z    +0.000, E1  +355.213, E3 -382386.405}
SPL {X  -159.990, Y  +656.991, Z    +0.000, E1  +350.742, E3 -382387.825}
SPL {X  -159.990, Y  +649.722, Z    +0.000, E1  +343.777, E3 -382390.743}
SPL {X  -159.990, Y  +645.752, Z    +0.000, E1  +340.157, E3 -382392.684}
SPL {X  -159.990, Y  +620.451, Z    +0.000, E1  +325.419, E3 -382415.401}
SPL {X  -159.990, Y  +591.256, Z    +0.000, E1  +319.966, E3 -382461.895}
SPL {X  -159.990, Y  +586.740, Z    +0.000, E1  +319.956, E3 -382473.285}
SPL {X  -159.990, Y  +581.814, Z    +0.000, E1  +319.956, E3 -382485.725}
SPL {X  -159.990, Y  +577.274, Z    +0.000, E1  +319.964, E3 -382497.202}
SPL {X  -159.990, Y  +572.933, Z    +0.000, E1  +319.959, E3 -382508.143}
SPL {X  -159.990, Y  +568.504, Z    +0.000, E1  +319.956, E3 -382519.306}
SPL {X  -159.990, Y  +563.189, Z    +0.000, E1  +319.932, E3 -382532.680}
SPL {X  -159.990, Y  +557.707, Z    +0.000, E1  +319.949, E3 -382546.535}
SPL {X  -159.990, Y  +552.104, Z    +0.000, E1  +319.922, E3 -382560.610}
SPL {X  -159.990, Y  +545.912, Z    +0.000, E1  +319.929, E3 -382576.259}
SPL {X  -159.990, Y  +540.054, Z    +0.000, E1  +319.939, E3 -382591.086}
SPL {X  -159.990, Y  +535.835, Z    +0.000, E1  +319.966, E3 -382601.767}
SPL {X  -159.990, Y  +530.667, Z    +0.000, E1  +319.910, E3 -382614.708}
SPL {X  -159.990, Y  +523.984, Z    +0.000, E1  +319.922, E3 -382631.574}
SPL {X  -159.990, Y  +496.806, Z    +0.000, E1  +312.216, E3 -382645.489}
SPL {X  -159.990, Y  +490.245, Z    +0.000, E1  +312.831, E3 -382662.020}
SPL {X  -159.990, Y  +486.737, Z    +0.000, E1  +313.729, E3 -382674.026}
SPL {X  -159.990, Y  +483.955, Z    +0.000, E1  +314.316, E3 -382683.318}
SPL {X  -159.990, Y  +480.580, Z    +0.000, E1  +315.242, E3 -382695.939}
SPL {X  -159.990, Y  +476.546, Z    +0.000, E1  +316.165, E3 -382710.234}
SPL {X  -159.990, Y  +473.377, Z    +0.000, E1  +316.953, E3 -382721.848}
SPL {X  -159.990, Y  +470.788, Z    +0.000, E1  +317.853, E3 -382733.262}
SPL {X  -159.990, Y  +467.944, Z    +0.000, E1  +318.635, E3 -382744.583}
SPL {X  -159.990, Y  +465.057, Z    +0.000, E1  +319.375, E3 -382756.148}
SPL {X  -159.990, Y  +461.409, Z    +0.000, E1  +319.848, E3 -382768.048}
SPL {X  -159.990, Y  +456.934, Z    +0.000, E1  +319.854, E3 -382779.323}
SPL {X  -159.990, Y  +452.940, Z    +0.000, E1  +319.854, E3 -382789.368}
SPL {X  -159.990, Y  +448.856, Z    +0.000, E1  +319.859, E3 -382799.651}
SPL {X  -159.990, Y  +444.973, Z    +0.000, E1  +319.856, E3 -382809.417}
SPL {X  -159.990, Y  +439.927, Z    +0.000, E1  +319.837, E3 -382822.073}
SPL {X  -159.990, Y  +435.246, Z    +0.000, E1  +319.853, E3 -382833.882}
SPL {X  -159.990, Y  +430.690, Z    +0.000, E1  +319.854, E3 -382845.344}
SPL {X  -159.990, Y  +426.145, Z    +0.000, E1  +319.853, E3 -382856.784}
SPL {X  -159.990, Y  +421.880, Z    +0.000, E1  +319.860, E3 -382867.517}
SPL {X  -159.990, Y  +416.246, Z    +0.000, E1  +319.819, E3 -382881.646}
SPL {X  -159.990, Y  +409.936, Z    +0.000, E1  +319.849, E3 -382897.582}
SPL {X  -159.990, Y  +404.988, Z    +0.000, E1  +319.861, E3 -382910.048}
SPL {X  -159.990, Y  +400.535, Z    +0.000, E1  +319.859, E3 -382921.246}
SPL {X  -159.990, Y  +396.024, Z    +0.000, E1  +319.860, E3 -382932.602}
SPL {X  -159.990, Y  +391.614, Z    +0.000, E1  +319.860, E3 -382943.696}
SPL {X  -159.990, Y  +387.212, Z    +0.000, E1  +319.859, E3 -382954.768}
SPL {X  -159.990, Y  +382.743, Z    +0.000, E1  +319.857, E3 -382966.009}
SPL {X  -159.925, Y  +377.946, Z    +0.000, E1  +319.864, E3 -382978.146}
SPL {X  -159.703, Y  +372.915, Z    +0.000, E1  +319.904, E3 -382991.046}
SPL {X  -159.358, Y  +368.290, Z    +0.000, E1  +319.961, E3 -383003.009}
SPL {X  -158.955, Y  +364.333, Z    +0.000, E1  +320.046, E3 -383013.411}
SPL {X  -158.270, Y  +359.106, Z    +0.000, E1  +320.118, E3 -383027.222}
SPL {X  -157.143, Y  +352.453, Z    +0.000, E1  +320.322, E3 -383045.153}
SPL {X  -156.148, Y  +347.650, Z    +0.000, E1  +320.549, E3 -383058.339}
SPL {X  -155.268, Y  +343.918, Z    +0.000, E1  +320.696, E3 -383068.620}
SPL {X  -153.936, Y  +338.906, Z    +0.000, E1  +320.911, E3 -383082.559}
SPL {X  -152.628, Y  +334.526, Z    +0.000, E1  +321.188, E3 -383094.961}
SPL {X  -151.010, Y  +329.654, Z    +0.000, E1  +326.674, E3 -383152.797}
ENDSPLINE

SPLINE
SPL {X  -157.513, Y  +354.453, Z    +0.000, E1  +340.941, E3 -383198.832}
SPL {X  -159.408, Y  +368.861, Z    +0.000, E1  +348.865, E3 -383208.254}
SPL {X  -159.941, Y  +378.532, Z    +0.000, E1  +354.551, E3 -383211.860}
SPL {X  -159.990, Y  +383.966, Z    +0.000, E1  +358.149, E3 -383213.312}
SPL {X  -159.990, Y  +388.001, Z    +0.000, E1  +361.086, E3 -383214.247}
SPL {X  -159.990, Y  +392.647, Z    +0.000, E1  +364.974, E3 -383215.386}
SPL {X  -159.990, Y  +397.943, Z    +0.000, E1  +369.963, E3 -383216.970}
SPL {X  -159.990, Y  +406.530, Z    +0.000, E1  +377.917, E3 -383220.868}
SPL {X  -159.990, Y  +429.014, Z    +0.000, E1  +392.438, E3 -383239.524}
SPL {X  -159.990, Y  +437.635, Z    +0.000, E1  +395.495, E3 -383249.757}
SPL {X  -159.990, Y  +460.330, Z    +0.000, E1  +398.908, E3 -383290.444}
SPL {X  -159.990, Y  +464.953, Z    +0.000, E1  +398.907, E3 -383302.602}
SPL {X  -159.990, Y  +469.353, Z    +0.000, E1  +398.902, E3 -383314.183}
SPL {X  -159.990, Y  +473.222, Z    +0.000, E1  +398.891, E3 -383324.391}
SPL {X  -159.990, Y  +477.957, Z    +0.000, E1  +398.922, E3 -383336.796}
SPL {X  -159.990, Y  +483.925, Z    +0.000, E1  +398.925, E3 -383352.466}
SPL {X  -159.990, Y  +489.893, Z    +0.000, E1  +398.930, E3 -383368.123}
SPL {X  -159.990, Y  +496.271, Z    +0.000, E1  +398.942, E3 -383384.880}
SPL {X  -159.990, Y  +502.093, Z    +0.000, E1  +398.909, E3 -383400.264}
SPL {X  -159.990, Y  +507.821, Z    +0.000, E1  +398.930, E3 -383415.284}
SPL {X  -159.990, Y  +513.533, Z    +0.000, E1  +398.910, E3 -383430.343}
SPL {X  -159.990, Y  +518.435, Z    +0.000, E1  +398.905, E3 -383443.238}
SPL {X  -159.990, Y  +523.478, Z    +0.000, E1  +398.918, E3 -383456.467}
SPL {X  -159.990, Y  +528.627, Z    +0.000, E1  +398.910, E3 -383470.020}
SPL {X  -159.990, Y  +533.053, Z    +0.000, E1  +398.899, E3 -383481.678}
SPL {X  -159.990, Y  +537.174, Z    +0.000, E1  +398.910, E3 -383492.492}
SPL {X  -159.990, Y  +541.259, Z    +0.000, E1  +398.888, E3 -383503.292}
SPL {X  -159.990, Y  +545.676, Z    +0.000, E1  +398.913, E3 -383514.863}
SPL {X  -159.990, Y  +550.777, Z    +0.000, E1  +398.906, E3 -383528.282}
SPL {X  -159.990, Y  +556.271, Z    +0.000, E1  +398.927, E3 -383542.685}
SPL {X  -159.990, Y  +561.696, Z    +0.000, E1  +398.912, E3 -383556.954}
SPL {X  -159.990, Y  +566.650, Z    +0.000, E1  +398.917, E3 -383569.968}
SPL {X  -159.990, Y  +571.814, Z    +0.000, E1  +398.914, E3 -383583.570}
SPL {X  -159.990, Y  +577.636, Z    +0.000, E1  +398.929, E3 -383598.868}
SPL {X  -159.990, Y  +583.167, Z    +0.000, E1  +398.906, E3 -383613.443}
SPL {X  -159.990, Y  +587.761, Z    +0.000, E1  +398.902, E3 -383625.528}
SPL {X  -159.990, Y  +592.962, Z    +0.000, E1  +398.925, E3 -383639.172}
SPL {X  -159.990, Y  +597.767, Z    +0.000, E1  +398.897, E3 -383651.848}
SPL {X  -159.990, Y  +602.727, Z    +0.000, E1  +398.920, E3 -383664.859}
SPL {X  -159.990, Y  +608.112, Z    +0.000, E1  +398.911, E3 -383679.033}
SPL {X  -159.990, Y  +614.125, Z    +0.000, E1  +398.936, E3 -383694.808}
SPL {X  -159.990, Y  +619.061, Z    +0.000, E1  +398.894, E3 -383707.840}
SPL {X  -159.990, Y  +623.264, Z    +0.000, E1  +398.906, E3 -383718.889}
SPL {X  -159.990, Y  +627.067, Z    +0.000, E1  +398.891, E3 -383728.909}
SPL {X  -159.990, Y  +630.187, Z    +0.000, E1  +398.892, E3 -383737.096}
SPL {X  -159.990, Y  +634.089, Z    +0.000, E1  +398.907, E3 -383747.333}
SPL {X  -159.990, Y  +638.639, Z    +0.000, E1  +398.904, E3 -383759.318}
SPL {X  -159.990, Y  +643.555, Z    +0.000, E1  +398.910, E3 -383772.238}
SPL {X  -159.990, Y  +649.380, Z    +0.000, E1  +398.930, E3 -383787.516}
SPL {X  -159.990, Y  +654.813, Z    +0.000, E1  +398.905, E3 -383801.840}
SPL {X  -159.990, Y  +658.715, Z    +0.000, E1  +398.892, E3 -383812.121}
SPL {X  -159.990, Y  +661.848, Z    +0.000, E1  +398.892, E3 -383820.360}
SPL {X  -159.990, Y  +665.703, Z    +0.000, E1  +398.903, E3 -383830.479}
SPL {X  -159.990, Y  +669.966, Z    +0.000, E1  +398.902, E3 -383841.685}
SPL {X  -159.954, Y  +674.895, Z    +0.000, E1  +398.910, E3 -383854.665}
SPL {X  -159.761, Y  +680.061, Z    +0.000, E1  +398.873, E3 -383868.444}
SPL {X  -159.443, Y  +684.716, Z    +0.000, E1  +398.815, E3 -383881.009}
SPL {X  -158.962, Y  +689.604, Z    +0.000, E1  +398.740, E3 -383894.379}
SPL {X  -158.318, Y  +694.567, Z    +0.000, E1  +398.614, E3 -383908.140}
SPL {X  -157.472, Y  +699.775, Z    +0.000, E1  +398.483, E3 -383922.699}
SPL {X  -156.506, Y  +704.705, Z    +0.000, E1  +398.294, E3 -383936.700}
SPL {X  -155.680, Y  +708.387, Z    +0.000, E1  +398.127, E3 -383947.271}
SPL {X  -154.586, Y  +712.730, Z    +0.000, E1  +397.967, E3 -383959.768}
SPL {X  -153.345, Y  +717.131, Z    +0.000, E1  +397.713, E3 -383972.652}
SPL {X  -151.080, Y  +724.146, Z    +0.000, E1  +393.201, E3 -384031.105}
ENDSPLINE

SPLINE
SPL {X  -157.921, Y  +697.149, Z    +0.000, E1  +377.701, E3 -384082.666}
SPL {X  -159.579, Y  +682.959, Z    +0.000, E1  +369.793, E3 -384090.615}
SPL {X  -159.938, Y  +675.561, Z    +0.000, E1  +365.399, E3 -384093.037}
SPL {X  -159.990, Y  +669.910, Z    +0.000, E1  +361.710, E3 -384094.328}
SPL {X  -159.990, Y  +665.465, Z    +0.000, E1  +358.378, E3 -384095.245}
SPL {X  -159.990, Y  +661.791, Z    +0.000, E1  +355.213, E3 -384096.083}
SPL {X  -159.990, Y  +656.991, Z    +0.000, E1  +350.742, E3 -384097.502}
SPL {X  -159.990, Y  +648.067, Z    +0.000, E1  +342.328, E3 -384101.232}
SPL {X  -159.990, Y  +620.451, Z    +0.000, E1  +325.419, E3 -384125.079}
SPL {X  -159.990, Y  +591.256, Z    +0.000, E1  +319.966, E3 -384171.572}
SPL {X  -159.990, Y  +586.740, Z    +0.000, E1  +319.956, E3 -384182.963}
SPL {X  -159.990, Y  +581.814, Z    +0.000, E1  +319.956, E3 -384195.402}
SPL {X  -159.990, Y  +577.274, Z    +0.000, E1  +319.964, E3 -384206.880}
SPL {X  -159.990, Y  +572.933, Z    +0.000, E1  +319.959, E3 -384217.821}
SPL {X  -159.990, Y  +568.504, Z    +0.000, E1  +319.956, E3 -384228.983}
SPL {X  -159.990, Y  +563.189, Z    +0.000, E1  +319.932, E3 -384242.357}
SPL {X  -159.990, Y  +557.707, Z    +0.000, E1  +319.949, E3 -384256.212}
SPL {X  -159.990, Y  +552.104, Z    +0.000, E1  +319.922, E3 -384270.287}
SPL {X  -159.990, Y  +545.912, Z    +0.000, E1  +319.929, E3 -384285.937}
SPL {X  -159.990, Y  +541.567, Z    +0.000, E1  +319.969, E3 -384296.991}
SPL {X  -159.990, Y  +537.213, Z    +0.000, E1  +319.937, E3 -384307.927}
SPL {X  -159.990, Y  +532.291, Z    +0.000, E1  +319.951, E3 -384320.352}
SPL {X  -159.990, Y  +527.393, Z    +0.000, E1  +319.924, E3 -384332.661}
SPL {X  -159.990, Y  +522.533, Z    +0.000, E1  +319.951, E3 -384344.959}
SPL {X  -159.990, Y  +502.378, Z    +0.000, E1  +313.079, E3 -384349.363}
SPL {X  -159.990, Y  +493.568, Z    +0.000, E1  +312.053, E3 -384360.530}
SPL {X  -159.990, Y  +489.464, Z    +0.000, E1  +313.059, E3 -384374.397}
SPL {X  -159.990, Y  +484.831, Z    +0.000, E1  +314.066, E3 -384389.930}
SPL {X  -159.990, Y  +480.580, Z    +0.000, E1  +315.242, E3 -384405.617}
SPL {X  -159.990, Y  +476.546, Z    +0.000, E1  +316.165, E3 -384419.911}
SPL {X  -159.990, Y  +473.377, Z    +0.000, E1  +316.953, E3 -384431.526}
SPL {X  -159.990, Y  +470.788, Z    +0.000, E1  +317.853, E3 -384442.939}
SPL {X  -159.990, Y  +467.944, Z    +0.000, E1  +318.635, E3 -384454.260}
SPL {X  -159.990, Y  +465.057, Z    +0.000, E1  +319.375, E3 -384465.826}
SPL {X  -159.990, Y  +461.409, Z    +0.000, E1  +319.848, E3 -384477.725}
SPL {X  -159.990, Y  +456.934, Z    +0.000, E1  +319.854, E3 -384489.001}
SPL {X  -159.990, Y  +452.940, Z    +0.000, E1  +319.854, E3 -384499.045}
SPL {X  -159.990, Y  +448.856, Z    +0.000, E1  +319.859, E3 -384509.329}
SPL {X  -159.990, Y  +444.973, Z    +0.000, E1  +319.856, E3 -384519.094}
SPL {X  -159.990, Y  +439.927, Z    +0.000, E1  +319.837, E3 -384531.750}
SPL {X  -159.990, Y  +435.246, Z    +0.000, E1  +319.853, E3 -384543.560}
SPL {X  -159.990, Y  +430.690, Z    +0.000, E1  +319.854, E3 -384555.022}
SPL {X  -159.990, Y  +426.145, Z    +0.000, E1  +319.853, E3 -384566.461}
SPL {X  -159.990, Y  +421.880, Z    +0.000, E1  +319.860, E3 -384577.194}
SPL {X  -159.990, Y  +416.246, Z    +0.000, E1  +319.819, E3 -384591.323}
SPL {X  -159.990, Y  +409.936, Z    +0.000, E1  +319.849, E3 -384607.260}
SPL {X  -159.990, Y  +404.988, Z    +0.000, E1  +319.861, E3 -384619.725}
SPL {X  -159.990, Y  +400.535, Z    +0.000, E1  +319.859, E3 -384630.923}
SPL {X  -159.990, Y  +396.024, Z    +0.000, E1  +319.860, E3 -384642.279}
SPL {X  -159.990, Y  +391.614, Z    +0.000, E1  +319.860, E3 -384653.373}
SPL {X  -159.990, Y  +387.212, Z    +0.000, E1  +319.859, E3 -384664.445}
SPL {X  -159.990, Y  +382.743, Z    +0.000, E1  +319.857, E3 -384675.687}
SPL {X  -159.925, Y  +377.946, Z    +0.000, E1  +319.864, E3 -384687.824}
SPL {X  -159.703, Y  +372.915, Z    +0.000, E1  +319.904, E3 -384700.723}
SPL {X  -159.358, Y  +368.290, Z    +0.000, E1  +319.961, E3 -384712.686}
SPL {X  -158.955, Y  +364.333, Z    +0.000, E1  +320.046, E3 -384723.089}
SPL {X  -158.482, Y  +360.589, Z    +0.000, E1  +320.125, E3 -384733.015}
SPL {X  -157.729, Y  +355.695, Z    +0.000, E1  +320.237, E3 -384746.087}
SPL {X  -156.893, Y  +351.173, Z    +0.000, E1  +320.410, E3 -384758.371}
SPL {X  -156.148, Y  +347.650, Z    +0.000, E1  +320.549, E3 -384768.017}
SPL {X  -155.268, Y  +343.918, Z    +0.000, E1  +320.696, E3 -384778.297}
SPL {X  -154.153, Y  +339.677, Z    +0.000, E1  +320.896, E3 -384790.104}
SPL {X  -152.885, Y  +335.352, Z    +0.000, E1  +321.114, E3 -384802.258}
SPL {X  -151.010, Y  +329.654, Z    +0.000, E1  +326.674, E3 -384862.475}
ENDSPLINE

SPLINE
SPL {X  -157.513, Y  +354.453, Z    +0.000, E1  +340.941, E3 -384908.509}
SPL {X  -159.408, Y  +368.861, Z    +0.000, E1  +348.865, E3 -384917.932}
SPL {X  -159.941, Y  +378.532, Z    +0.000, E1  +354.551, E3 -384921.537}
SPL {X  -159.990, Y  +383.966, Z    +0.000, E1  +358.149, E3 -384922.989}
SPL {X  -159.990, Y  +388.001, Z    +0.000, E1  +361.086, E3 -384923.924}
SPL {X  -159.990, Y  +392.647, Z    +0.000, E1  +364.974, E3 -384925.063}
SPL {X  -159.990, Y  +397.943, Z    +0.000, E1  +369.963, E3 -384926.648}
SPL {X  -159.990, Y  +406.530, Z    +0.000, E1  +377.917, E3 -384930.545}
SPL {X  -159.990, Y  +429.014, Z    +0.000, E1  +392.438, E3 -384949.202}
SPL {X  -159.990, Y  +437.635, Z    +0.000, E1  +395.495, E3 -384959.434}
SPL {X  -159.990, Y  +460.330, Z    +0.000, E1  +398.908, E3 -385000.121}
SPL {X  -159.990, Y  +464.953, Z    +0.000, E1  +398.907, E3 -385012.280}
SPL {X  -159.990, Y  +469.353, Z    +0.000, E1  +398.902, E3 -385023.860}
SPL {X  -159.990, Y  +473.222, Z    +0.000, E1  +398.891, E3 -385034.069}
SPL {X  -159.990, Y  +476.615, Z    +0.000, E1  +398.890, E3 -385043.003}
SPL {X  -159.990, Y  +481.308, Z    +0.000, E1  +398.917, E3 -385055.286}
SPL {X  -159.990, Y  +486.996, Z    +0.000, E1  +398.928, E3 -385070.194}
SPL {X  -159.990, Y  +491.333, Z    +0.000, E1  +398.896, E3 -385081.634}
SPL {X  -159.990, Y  +496.271, Z    +0.000, E1  +398.942, E3 -385094.557}
SPL {X  -159.990, Y  +502.093, Z    +0.000, E1  +398.909, E3 -385109.941}
SPL {X  -159.990, Y  +507.821, Z    +0.000, E1  +398.930, E3 -385124.961}
SPL {X  -159.990, Y  +513.533, Z    +0.000, E1  +398.910, E3 -385140.021}
SPL {X  -159.990, Y  +518.435, Z    +0.000, E1  +398.905, E3 -385152.916}
SPL {X  -159.990, Y  +523.478, Z    +0.000, E1  +398.918, E3 -385166.144}
SPL {X  -159.990, Y  +528.627, Z    +0.000, E1  +398.910, E3 -385179.698}
SPL {X  -159.990, Y  +533.053, Z    +0.000, E1  +398.899, E3 -385191.355}
SPL {X  -159.990, Y  +537.174, Z    +0.000, E1  +398.910, E3 -385202.170}
SPL {X  -159.990, Y  +542.636, Z    +0.000, E1  +398.920, E3 -385216.538}
SPL {X  -159.990, Y  +549.483, Z    +0.000, E1  +398.950, E3 -385234.493}
SPL {X  -159.990, Y  +554.638, Z    +0.000, E1  +398.890, E3 -385248.130}
SPL {X  -159.990, Y  +557.678, Z    +0.000, E1  +398.893, E3 -385256.106}
SPL {X  -159.990, Y  +561.696, Z    +0.000, E1  +398.912, E3 -385266.631}
SPL {X  -159.990, Y  +566.650, Z    +0.000, E1  +398.917, E3 -385279.645}
SPL {X  -159.990, Y  +571.814, Z    +0.000, E1  +398.914, E3 -385293.248}
SPL {X  -159.990, Y  +577.636, Z    +0.000, E1  +398.929, E3 -385308.545}
SPL {X  -159.990, Y  +583.167, Z    +0.000, E1  +398.906, E3 -385323.121}
SPL {X  -159.990, Y  +587.761, Z    +0.000, E1  +398.902, E3 -385335.206}
SPL {X  -159.990, Y  +592.962, Z    +0.000, E1  +398.925, E3 -385348.850}
SPL {X  -159.990, Y  +597.767, Z    +0.000, E1  +398.897, E3 -385361.525}
SPL {X  -159.990, Y  +602.727, Z    +0.000, E1  +398.920, E3 -385374.536}
SPL {X  -159.990, Y  +608.112, Z    +0.000, E1  +398.911, E3 -385388.710}
SPL {X  -159.990, Y  +613.039, Z    +0.000, E1  +398.906, E3 -385401.673}
SPL {X  -159.990, Y  +618.087, Z    +0.000, E1  +398.915, E3 -385414.932}
SPL {X  -159.990, Y  +623.264, Z    +0.000, E1  +398.906, E3 -385428.566}
SPL {X  -159.990, Y  +628.669, Z    +0.000, E1  +398.928, E3 -385442.734}
SPL {X  -159.990, Y  +634.089, Z    +0.000, E1  +398.907, E3 -385457.010}
SPL {X  -159.990, Y  +638.639, Z    +0.000, E1  +398.904, E3 -385468.996}
SPL {X  -159.990, Y  +644.750, Z    +0.000, E1  +398.946, E3 -385485.001}
SPL {X  -159.990, Y  +650.458, Z    +0.000, E1  +398.900, E3 -385500.073}
SPL {X  -159.990, Y  +654.813, Z    +0.000, E1  +398.905, E3 -385511.518}
SPL {X  -159.990, Y  +660.353, Z    +0.000, E1  +398.930, E3 -385526.049}
SPL {X  -159.990, Y  +665.703, Z    +0.000, E1  +398.903, E3 -385540.156}
SPL {X  -159.990, Y  +669.966, Z    +0.000, E1  +398.902, E3 -385551.363}
SPL {X  -159.954, Y  +674.895, Z    +0.000, E1  +398.910, E3 -385564.343}
SPL {X  -159.761, Y  +680.061, Z    +0.000, E1  +398.873, E3 -385578.122}
SPL {X  -159.327, Y  +686.045, Z    +0.000, E1  +398.835, E3 -385594.244}
SPL {X  -158.832, Y  +690.714, Z    +0.000, E1  +398.685, E3 -385607.170}
SPL {X  -158.318, Y  +694.567, Z    +0.000, E1  +398.614, E3 -385617.817}
SPL {X  -157.472, Y  +699.775, Z    +0.000, E1  +398.483, E3 -385632.377}
SPL {X  -156.506, Y  +704.705, Z    +0.000, E1  +398.294, E3 -385646.377}
SPL {X  -155.357, Y  +709.721, Z    +0.000, E1  +398.108, E3 -385660.732}
SPL {X  -154.286, Y  +713.838, Z    +0.000, E1  +397.877, E3 -385672.715}
SPL {X  -153.345, Y  +717.131, Z    +0.000, E1  +397.713, E3 -385682.329}
SPL {X  -151.080, Y  +724.146, Z    +0.000, E1  +393.201, E3 -385740.783}
ENDSPLINE

SPLINE
SPL {X  -157.921, Y  +697.149, Z    +0.000, E1  +377.701, E3 -385792.344}
SPL {X  -159.579, Y  +682.959, Z    +0.000, E1  +369.793, E3 -385800.292}
SPL {X  -159.938, Y  +675.561, Z    +0.000, E1  +365.399, E3 -385802.714}
SPL {X  -159.990, Y  +669.910, Z    +0.000, E1  +361.710, E3 -385804.005}
SPL {X  -159.990, Y  +665.465, Z    +0.000, E1  +358.378, E3 -385804.922}
SPL {X  -159.990, Y  +661.791, Z    +0.000, E1  +355.213, E3 -385805.760}
SPL {X  -159.990, Y  +656.991, Z    +0.000, E1  +350.742, E3 -385807.180}
SPL {X  -159.990, Y  +648.067, Z    +0.000, E1  +342.328, E3 -385810.909}
SPL {X  -159.990, Y  +620.451, Z    +0.000, E1  +325.419, E3 -385834.756}
SPL {X  -159.990, Y  +591.256, Z    +0.000, E1  +319.966, E3 -385881.250}
SPL {X  -159.990, Y  +586.740, Z    +0.000, E1  +319.956, E3 -385892.640}
SPL {X  -159.990, Y  +581.814, Z    +0.000, E1  +319.956, E3 -385905.080}
SPL {X  -159.990, Y  +577.274, Z    +0.000, E1  +319.964, E3 -385916.557}
SPL {X  -159.990, Y  +572.933, Z    +0.000, E1  +319.959, E3 -385927.498}
SPL {X  -159.990, Y  +568.504, Z    +0.000, E1  +319.956, E3 -385938.661}
SPL {X  -159.990, Y  +563.189, Z    +0.000, E1  +319.932, E3 -385952.034}
SPL {X  -159.990, Y  +557.707, Z    +0.000, E1  +319.949, E3 -385965.890}
SPL {X  -159.990, Y  +553.571, Z    +0.000, E1  +319.954, E3 -385976.308}
SPL {X  -159.990, Y  +549.413, Z    +0.000, E1  +319.938, E3 -385986.774}
SPL {X  -159.990, Y  +543.439, Z    +0.000, E1  +319.921, E3 -386001.862}
SPL {X  -159.990, Y  +537.213, Z    +0.000, E1  +319.937, E3 -386017.605}
SPL {X  -159.990, Y  +530.667, Z    +0.000, E1  +319.910, E3 -386034.062}
SPL {X  -159.990, Y  +523.984, Z    +0.000, E1  +319.922, E3 -386050.929}
SPL {X  -159.990, Y  +502.378, Z    +0.000, E1  +313.079, E3 -386059.040}
SPL {X  -159.990, Y  +493.568, Z    +0.000, E1  +312.053, E3 -386070.208}
SPL {X  -159.990, Y  +488.437, Z    +0.000, E1  +313.241, E3 -386087.423}
SPL {X  -159.990, Y  +483.955, Z    +0.000, E1  +314.316, E3 -386102.673}
SPL {X  -159.990, Y  +479.762, Z    +0.000, E1  +315.381, E3 -386118.064}
SPL {X  -159.990, Y  +474.562, Z    +0.000, E1  +316.600, E3 -386136.734}
SPL {X  -159.990, Y  +470.788, Z    +0.000, E1  +317.853, E3 -386152.617}
SPL {X  -159.990, Y  +467.944, Z    +0.000, E1  +318.635, E3 -386163.938}
SPL {X  -159.990, Y  +465.057, Z    +0.000, E1  +319.375, E3 -386175.503}
SPL {X  -159.990, Y  +461.409, Z    +0.000, E1  +319.848, E3 -386187.402}
SPL {X  -159.990, Y  +456.934, Z    +0.000, E1  +319.854, E3 -386198.678}
SPL {X  -159.990, Y  +452.940, Z    +0.000, E1  +319.854, E3 -386208.723}
SPL {X  -159.990, Y  +448.856, Z    +0.000, E1  +319.859, E3 -386219.006}
SPL {X  -159.990, Y  +443.741, Z    +0.000, E1  +319.827, E3 -386231.824}
SPL {X  -159.990, Y  +436.703, Z    +0.000, E1  +319.809, E3 -386249.506}
SPL {X  -159.990, Y  +430.690, Z    +0.000, E1  +319.854, E3 -386264.699}
SPL {X  -159.990, Y  +426.145, Z    +0.000, E1  +319.853, E3 -386276.139}
SPL {X  -159.990, Y  +421.880, Z    +0.000, E1  +319.860, E3 -386286.872}
SPL {X  -159.990, Y  +416.246, Z    +0.000, E1  +319.819, E3 -386301.000}
SPL {X  -159.990, Y  +409.936, Z    +0.000, E1  +319.849, E3 -386316.937}
SPL {X  -159.990, Y  +404.988, Z    +0.000, E1  +319.861, E3 -386329.403}
SPL {X  -159.990, Y  +400.535, Z    +0.000, E1  +319.859, E3 -386340.601}
SPL {X  -159.990, Y  +396.024, Z    +0.000, E1  +319.860, E3 -386351.957}
SPL {X  -159.990, Y  +391.614, Z    +0.000, E1  +319.860, E3 -386363.050}
SPL {X  -159.990, Y  +387.212, Z    +0.000, E1  +319.859, E3 -386374.123}
SPL {X  -159.990, Y  +382.743, Z    +0.000, E1  +319.857, E3 -386385.364}
SPL {X  -159.925, Y  +377.946, Z    +0.000, E1  +319.864, E3 -386397.501}
SPL {X  -159.703, Y  +372.915, Z    +0.000, E1  +319.904, E3 -386410.401}
SPL {X  -159.358, Y  +368.290, Z    +0.000, E1  +319.961, E3 -386422.363}
SPL {X  -158.955, Y  +364.333, Z    +0.000, E1  +320.046, E3 -386432.766}
SPL {X  -158.482, Y  +360.589, Z    +0.000, E1  +320.125, E3 -386442.692}
SPL {X  -157.729, Y  +355.695, Z    +0.000, E1  +320.237, E3 -386455.765}
SPL {X  -156.893, Y  +351.173, Z    +0.000, E1  +320.410, E3 -386468.048}
SPL {X  -156.148, Y  +347.650, Z    +0.000, E1  +320.549, E3 -386477.694}
SPL {X  -155.268, Y  +343.918, Z    +0.000, E1  +320.696, E3 -386487.975}
SPL {X  -154.153, Y  +339.677, Z    +0.000, E1  +320.896, E3 -386499.782}
SPL {X  -152.885, Y  +335.352, Z    +0.000, E1  +321.114, E3 -386511.936}
SPL {X  -151.010, Y  +329.654, Z    +0.000, E1  +326.674, E3 -386572.152}
ENDSPLINE

SPLINE
SPL {X  -157.513, Y  +354.453, Z    +0.000, E1  +340.941, E3 -386618.186}
SPL {X  -159.638, Y  +371.886, Z    +0.000, E1  +350.545, E3 -386628.849}
SPL {X  -159.990, Y  +382.357, Z    +0.000, E1  +356.972, E3 -386632.264}
SPL {X  -159.990, Y  +388.001, Z    +0.000, E1  +361.086, E3 -386633.602}
SPL {X  -159.990, Y  +392.647, Z    +0.000, E1  +364.974, E3 -386634.740}
SPL {X  -159.990, Y  +399.434, Z    +0.000, E1  +371.306, E3 -386636.921}
SPL {X  -159.990, Y  +409.375, Z    +0.000, E1  +380.357, E3 -386641.953}
SPL {X  -159.990, Y  +434.822, Z    +0.000, E1  +394.625, E3 -386665.523}
SPL {X  -159.990, Y  +460.330, Z    +0.000, E1  +398.908, E3 -386709.799}
SPL {X  -159.990, Y  +464.953, Z    +0.000, E1  +398.907, E3 -386721.957}
SPL {X  -159.990, Y  +469.353, Z    +0.000, E1  +398.902, E3 -386733.537}
SPL {X  -159.990, Y  +475.034, Z    +0.000, E1  +398.936, E3 -386748.453}
SPL {X  -159.990, Y  +481.308, Z    +0.000, E1  +398.917, E3 -386764.963}
SPL {X  -159.990, Y  +485.396, Z    +0.000, E1  +398.893, E3 -386775.723}
SPL {X  -159.990, Y  +488.362, Z    +0.000, E1  +398.896, E3 -386783.506}
SPL {X  -159.990, Y  +492.629, Z    +0.000, E1  +398.922, E3 -386794.678}
SPL {X  -159.990, Y  +497.431, Z    +0.000, E1  +398.905, E3 -386807.344}
SPL {X  -159.990, Y  +502.093, Z    +0.000, E1  +398.909, E3 -386819.618}
SPL {X  -159.990, Y  +507.821, Z    +0.000, E1  +398.930, E3 -386834.639}
SPL {X  -159.990, Y  +513.533, Z    +0.000, E1  +398.910, E3 -386849.698}
SPL {X  -159.990, Y  +518.435, Z    +0.000, E1  +398.905, E3 -386862.593}
SPL {X  -159.990, Y  +523.478, Z    +0.000, E1  +398.918, E3 -386875.822}
SPL {X  -159.990, Y  +528.627, Z    +0.000, E1  +398.910, E3 -386889.375}
SPL {X  -159.990, Y  +533.053, Z    +0.000, E1  +398.899, E3 -386901.033}
SPL {X  -159.990, Y  +537.174, Z    +0.000, E1  +398.910, E3 -386911.847}
SPL {X  -159.990, Y  +541.259, Z    +0.000, E1  +398.888, E3 -386922.647}
SPL {X  -159.990, Y  +545.676, Z    +0.000, E1  +398.913, E3 -386934.218}
SPL {X  -159.990, Y  +550.777, Z    +0.000, E1  +398.906, E3 -386947.637}
SPL {X  -159.990, Y  +554.638, Z    +0.000, E1  +398.890, E3 -386957.807}
SPL {X  -159.990, Y  +557.678, Z    +0.000, E1  +398.893, E3 -386965.783}
SPL {X  -159.990, Y  +561.696, Z    +0.000, E1  +398.912, E3 -386976.309}
SPL {X  -159.990, Y  +566.650, Z    +0.000, E1  +398.917, E3 -386989.323}
SPL {X  -159.990, Y  +571.814, Z    +0.000, E1  +398.914, E3 -387002.925}
SPL {X  -159.990, Y  +577.636, Z    +0.000, E1  +398.929, E3 -387018.223}
SPL {X  -159.990, Y  +583.167, Z    +0.000, E1  +398.906, E3 -387032.798}
SPL {X  -159.990, Y  +587.761, Z    +0.000, E1  +398.902, E3 -387044.883}
SPL {X  -159.990, Y  +592.962, Z    +0.000, E1  +398.925, E3 -387058.527}
SPL {X  -159.990, Y  +597.767, Z    +0.000, E1  +398.897, E3 -387071.202}
SPL {X  -159.990, Y  +602.727, Z    +0.000, E1  +398.920, E3 -387084.213}
SPL {X  -159.990, Y  +608.112, Z    +0.000, E1  +398.911, E3 -387098.388}
SPL {X  -159.990, Y  +614.125, Z    +0.000, E1  +398.936, E3 -387114.163}
SPL {X  -159.990, Y  +619.061, Z    +0.000, E1  +398.894, E3 -387127.194}
SPL {X  -159.990, Y  +623.264, Z    +0.000, E1  +398.906, E3 -387138.243}
SPL {X  -159.990, Y  +628.669, Z    +0.000, E1  +398.928, E3 -387152.412}
SPL {X  -159.990, Y  +634.089, Z    +0.000, E1  +398.907, E3 -387166.687}
SPL {X  -159.990, Y  +638.639, Z    +0.000, E1  +398.904, E3 -387178.673}
SPL {X  -159.990, Y  +643.555, Z    +0.000, E1  +398.910, E3 -387191.593}
SPL {X  -159.990, Y  +649.380, Z    +0.000, E1  +398.930, E3 -387206.870}
SPL {X  -159.990, Y  +654.813, Z    +0.000, E1  +398.905, E3 -387221.195}
SPL {X  -159.990, Y  +660.353, Z    +0.000, E1  +398.930, E3 -387235.726}
SPL {X  -159.990, Y  +665.703, Z    +0.000, E1  +398.903, E3 -387249.834}
SPL {X  -159.990, Y  +671.472, Z    +0.000, E1  +398.942, E3 -387264.938}
SPL {X  -159.920, Y  +676.216, Z    +0.000, E1  +398.875, E3 -387277.573}
SPL {X  -159.761, Y  +680.061, Z    +0.000, E1  +398.873, E3 -387287.799}
SPL {X  -159.443, Y  +684.716, Z    +0.000, E1  +398.815, E3 -387300.364}
SPL {X  -158.962, Y  +689.604, Z    +0.000, E1  +398.740, E3 -387313.734}
SPL {X  -158.318, Y  +694.567, Z    +0.000, E1  +398.614, E3 -387327.495}
SPL {X  -157.472, Y  +699.775, Z    +0.000, E1  +398.483, E3 -387342.054}
SPL {X  -156.506, Y  +704.705, Z    +0.000, E1  +398.294, E3 -387356.055}
SPL {X  -155.357, Y  +709.721, Z    +0.000, E1  +398.108, E3 -387370.410}
SPL {X  -154.286, Y  +713.838, Z    +0.000, E1  +397.877, E3 -387382.392}
SPL {X  -153.345, Y  +717.131, Z    +0.000, E1  +397.713, E3 -387392.007}
SPL {X  -151.080, Y  +724.146, Z    +0.000, E1  +393.201, E3 -387450.460}
ENDSPLINE

SPLINE
SPL {X  -157.921, Y  +697.149, Z    +0.000, E1  +377.701, E3 -387502.021}
SPL {X  -159.579, Y  +682.959, Z    +0.000, E1  +369.793, E3 -387509.969}
SPL {X  -159.938, Y  +675.561, Z    +0.000, E1  +365.399, E3 -387512.392}
SPL {X  -159.990, Y  +669.910, Z    +0.000, E1  +361.710, E3 -387513.682}
SPL {X  -159.990, Y  +665.465, Z    +0.000, E1  +358.378, E3 -387514.600}
SPL {X  -159.990, Y  +661.791, Z    +0.000, E1  +355.213, E3 -387515.438}
SPL {X  -159.990, Y  +656.991, Z    +0.000, E1  +350.742, E3 -387516.857}
SPL {X  -159.990, Y  +649.722, Z    +0.000, E1  +343.777, E3 -387519.775}
SPL {X  -159.990, Y  +645.752, Z    +0.000, E1  +340.157, E3 -387521.717}
SPL {X  -159.990, Y  +624.891, Z    +0.000, E1  +327.004, E3 -387539.074}
SPL {X  -159.990, Y  +618.109, Z    +0.000, E1  +324.631, E3 -387547.250}
SPL {X  -159.990, Y  +591.256, Z    +0.000, E1  +319.966, E3 -387590.927}
SPL {X  -159.990, Y  +586.740, Z    +0.000, E1  +319.956, E3 -387602.317}
SPL {X  -159.990, Y  +581.814, Z    +0.000, E1  +319.956, E3 -387614.757}
SPL {X  -159.990, Y  +577.274, Z    +0.000, E1  +319.964, E3 -387626.234}
SPL {X  -159.990, Y  +572.933, Z    +0.000, E1  +319.959, E3 -387637.176}
SPL {X  -159.990, Y  +568.504, Z    +0.000, E1  +319.956, E3 -387648.338}
SPL {X  -159.990, Y  +564.427, Z    +0.000, E1  +319.959, E3 -387658.624}
SPL {X  -159.990, Y  +558.823, Z    +0.000, E1  +319.916, E3 -387672.704}
SPL {X  -159.990, Y  +553.571, Z    +0.000, E1  +319.954, E3 -387685.985}
SPL {X  -159.990, Y  +549.413, Z    +0.000, E1  +319.938, E3 -387696.452}
SPL {X  -159.990, Y  +544.924, Z    +0.000, E1  +319.955, E3 -387707.833}
SPL {X  -159.990, Y  +540.054, Z    +0.000, E1  +319.939, E3 -387720.119}
SPL {X  -159.990, Y  +533.683, Z    +0.000, E1  +319.916, E3 -387736.143}
SPL {X  -159.990, Y  +528.899, Z    +0.000, E1  +319.955, E3 -387748.260}
SPL {X  -159.990, Y  +523.984, Z    +0.000, E1  +319.922, E3 -387760.606}
SPL {X  -159.990, Y  +495.402, Z    +0.000, E1  +312.238, E3 -387777.536}
SPL {X  -159.990, Y  +489.464, Z    +0.000, E1  +313.059, E3 -387793.752}
SPL {X  -159.990, Y  +484.831, Z    +0.000, E1  +314.066, E3 -387809.285}
SPL {X  -159.990, Y  +480.580, Z    +0.000, E1  +315.242, E3 -387824.971}
SPL {X  -159.990, Y  +476.546, Z    +0.000, E1  +316.165, E3 -387839.266}
SPL {X  -159.990, Y  +473.377, Z    +0.000, E1  +316.953, E3 -387850.881}
SPL {X  -159.990, Y  +470.788, Z    +0.000, E1  +317.853, E3 -387862.294}
SPL {X  -159.990, Y  +467.944, Z    +0.000, E1  +318.635, E3 -387873.615}
SPL {X  -159.990, Y  +465.057, Z    +0.000, E1  +319.375, E3 -387885.180}
SPL {X  -159.990, Y  +461.409, Z    +0.000, E1  +319.848, E3 -387897.080}
SPL {X  -159.990, Y  +456.934, Z    +0.000, E1  +319.854, E3 -387908.356}
SPL {X  -159.990, Y  +452.940, Z    +0.000, E1  +319.854, E3 -387918.400}
SPL {X  -159.990, Y  +448.856, Z    +0.000, E1  +319.859, E3 -387928.683}
SPL {X  -159.990, Y  +444.973, Z    +0.000, E1  +319.856, E3 -387938.449}
SPL {X  -159.990, Y  +439.927, Z    +0.000, E1  +319.837, E3 -387951.105}
SPL {X  -159.990, Y  +435.246, Z    +0.000, E1  +319.853, E3 -387962.915}
SPL {X  -159.990, Y  +430.690, Z    +0.000, E1  +319.854, E3 -387974.376}
SPL {X  -159.990, Y  +426.145, Z    +0.000, E1  +319.853, E3 -387985.816}
SPL {X  -159.990, Y  +421.880, Z    +0.000, E1  +319.860, E3 -387996.549}
SPL {X  -159.990, Y  +416.246, Z    +0.000, E1  +319.819, E3 -388010.678}
SPL {X  -159.990, Y  +409.936, Z    +0.000, E1  +319.849, E3 -388026.615}
SPL {X  -159.990, Y  +404.988, Z    +0.000, E1  +319.861, E3 -388039.080}
SPL {X  -159.990, Y  +400.535, Z    +0.000, E1  +319.859, E3 -388050.278}
SPL {X  -159.990, Y  +396.024, Z    +0.000, E1  +319.860, E3 -388061.634}
SPL {X  -159.990, Y  +391.614, Z    +0.000, E1  +319.860, E3 -388072.728}
SPL {X  -159.990, Y  +387.212, Z    +0.000, E1  +319.859, E3 -388083.800}
SPL {X  -159.990, Y  +382.743, Z    +0.000, E1  +319.857, E3 -388095.042}
SPL {X  -159.925, Y  +377.946, Z    +0.000, E1  +319.864, E3 -388107.179}
SPL {X  -159.703, Y  +372.915, Z    +0.000, E1  +319.904, E3 -388120.078}
SPL {X  -159.358, Y  +368.290, Z    +0.000, E1  +319.961, E3 -388132.041}
SPL {X  -158.955, Y  +364.333, Z    +0.000, E1  +320.046, E3 -388142.443}
SPL {X  -158.270, Y  +359.106, Z    +0.000, E1  +320.118, E3 -388156.254}
SPL {X  -157.143, Y  +352.453, Z    +0.000, E1  +320.322, E3 -388174.185}
SPL {X  -156.148, Y  +347.650, Z    +0.000, E1  +320.549, E3 -388187.372}
SPL {X  -155.268, Y  +343.918, Z    +0.000, E1  +320.696, E3 -388197.652}
SPL {X  -153.936, Y  +338.906, Z    +0.000, E1  +320.911, E3 -388211.592}
SPL {X  -152.628, Y  +334.526, Z    +0.000, E1  +321.188, E3 -388223.994}
SPL {X  -151.010, Y  +329.654, Z    +0.000, E1  +326.674, E3 -388281.830}
ENDSPLINE

SPLINE
SPL {X  -157.513, Y  +354.453, Z    +0.000, E1  +340.941, E3 -388327.864}
SPL {X  -159.408, Y  +368.861, Z    +0.000, E1  +348.865, E3 -388337.287}
SPL {X  -159.941, Y  +378.532, Z    +0.000, E1  +354.551, E3 -388340.892}
SPL {X  -159.990, Y  +383.966, Z    +0.000, E1  +358.149, E3 -388342.344}
SPL {X  -159.990, Y  +389.165, Z    +0.000, E1  +361.929, E3 -388343.546}
SPL {X  -159.990, Y  +394.164, Z    +0.000, E1  +366.430, E3 -388344.838}
SPL {X  -159.990, Y  +399.434, Z    +0.000, E1  +371.306, E3 -388346.598}
SPL {X  -159.990, Y  +407.956, Z    +0.000, E1  +379.215, E3 -388350.686}
SPL {X  -159.990, Y  +429.014, Z    +0.000, E1  +392.438, E3 -388368.557}
SPL {X  -159.990, Y  +437.635, Z    +0.000, E1  +395.495, E3 -388378.789}
SPL {X  -159.990, Y  +460.330, Z    +0.000, E1  +398.908, E3 -388419.476}
SPL {X  -159.990, Y  +464.953, Z    +0.000, E1  +398.907, E3 -388431.635}
SPL {X  -159.990, Y  +469.353, Z    +0.000, E1  +398.902, E3 -388443.215}
SPL {X  -159.990, Y  +475.034, Z    +0.000, E1  +398.936, E3 -388458.130}
SPL {X  -159.990, Y  +481.308, Z    +0.000, E1  +398.917, E3 -388474.641}
SPL {X  -159.990, Y  +486.996, Z    +0.000, E1  +398.928, E3 -388489.548}
SPL {X  -159.990, Y  +492.629, Z    +0.000, E1  +398.922, E3 -388504.355}
SPL {X  -159.990, Y  +497.431, Z    +0.000, E1  +398.905, E3 -388517.021}
SPL {X  -159.990, Y  +502.093, Z    +0.000, E1  +398.909, E3 -388529.296}
SPL {X  -159.990, Y  +507.821, Z    +0.000, E1  +398.930, E3 -388544.316}
SPL {X  -159.990, Y  +513.533, Z    +0.000, E1  +398.910, E3 -388559.375}
SPL {X  -159.990, Y  +519.462, Z    +0.000, E1  +398.933, E3 -388574.928}
SPL {X  -159.990, Y  +524.415, Z    +0.000, E1  +398.896, E3 -388587.992}
SPL {X  -159.990, Y  +528.627, Z    +0.000, E1  +398.910, E3 -388599.053}
SPL {X  -159.990, Y  +533.053, Z    +0.000, E1  +398.899, E3 -388610.710}
SPL {X  -159.990, Y  +537.174, Z    +0.000, E1  +398.910, E3 -388621.525}
SPL {X  -159.990, Y  +541.259, Z    +0.000, E1  +398.888, E3 -388632.325}
SPL {X  -159.990, Y  +545.676, Z    +0.000, E1  +398.913, E3 -388643.895}
SPL {X  -159.990, Y  +550.777, Z    +0.000, E1  +398.906, E3 -388657.314}
SPL {X  -159.990, Y  +556.271, Z    +0.000, E1  +398.927, E3 -388671.717}
SPL {X  -159.990, Y  +561.696, Z    +0.000, E1  +398.912, E3 -388685.986}
SPL {X  -159.990, Y  +566.650, Z    +0.000, E1  +398.917, E3 -388699.000}
SPL {X  -159.990, Y  +571.814, Z    +0.000, E1  +398.914, E3 -388712.603}
SPL {X  -159.990, Y  +577.636, Z    +0.000, E1  +398.929, E3 -388727.900}
SPL {X  -159.990, Y  +583.167, Z    +0.000, E1  +398.906, E3 -388742.476}
SPL {X  -159.990, Y  +587.761, Z    +0.000, E1  +398.902, E3 -388754.560}
SPL {X  -159.990, Y  +592.962, Z    +0.000, E1  +398.925, E3 -388768.205}
SPL {X  -159.990, Y  +599.478, Z    +0.000, E1  +398.941, E3 -388785.315}
SPL {X  -159.990, Y  +606.904, Z    +0.000, E1  +398.953, E3 -388804.828}
SPL {X  -159.990, Y  +613.039, Z    +0.000, E1  +398.906, E3 -388821.028}
SPL {X  -159.990, Y  +618.087, Z    +0.000, E1  +398.915, E3 -388834.286}
SPL {X  -159.990, Y  +623.264, Z    +0.000, E1  +398.906, E3 -388847.921}
SPL {X  -159.990, Y  +628.669, Z    +0.000, E1  +398.928, E3 -388862.089}
SPL {X  -159.990, Y  +634.089, Z    +0.000, E1  +398.907, E3 -388876.365}
SPL {X  -159.990, Y  +638.639, Z    +0.000, E1  +398.904, E3 -388888.350}
SPL {X  -159.990, Y  +643.555, Z    +0.000, E1  +398.910, E3 -388901.270}
SPL {X  -159.990, Y  +649.380, Z    +0.000, E1  +398.930, E3 -388916.548}
SPL {X  -159.990, Y  +654.813, Z    +0.000, E1  +398.905, E3 -388930.872}
SPL {X  -159.990, Y  +660.353, Z    +0.000, E1  +398.930, E3 -388945.404}
SPL {X  -159.990, Y  +665.703, Z    +0.000, E1  +398.903, E3 -388959.511}
SPL {X  -159.990, Y  +671.472, Z    +0.000, E1  +398.942, E3 -388974.616}
SPL {X  -159.920, Y  +676.216, Z    +0.000, E1  +398.875, E3 -388987.251}
SPL {X  -159.761, Y  +680.061, Z    +0.000, E1  +398.873, E3 -388997.477}
SPL {X  -159.443, Y  +684.716, Z    +0.000, E1  +398.815, E3 -389010.042}
SPL {X  -158.962, Y  +689.604, Z    +0.000, E1  +398.740, E3 -389023.411}
SPL {X  -158.318, Y  +694.567, Z    +0.000, E1  +398.614, E3 -389037.172}
SPL {X  -157.472, Y  +699.775, Z    +0.000, E1  +398.483, E3 -389051.732}
SPL {X  -156.506, Y  +704.705, Z    +0.000, E1  +398.294, E3 -389065.732}
SPL {X  -155.680, Y  +708.387, Z    +0.000, E1  +398.127, E3 -389076.303}
SPL {X  -154.586, Y  +712.730, Z    +0.000, E1  +397.967, E3 -389088.800}
SPL {X  -153.345, Y  +717.131, Z    +0.000, E1  +397.713, E3 -389101.684}
SPL {X  -151.080, Y  +724.146, Z    +0.000, E1  +393.201, E3 -389160.138}
ENDSPLINE

SPLINE
SPL {X  -157.921, Y  +697.149, Z    +0.000, E1  +377.701, E3 -389211.699}
SPL {X  -159.579, Y  +682.959, Z    +0.000, E1  +369.793, E3 -389219.647}
SPL {X  -159.938, Y  +675.561, Z    +0.000, E1  +365.399, E3 -389222.069}
SPL {X  -159.990, Y  +669.910, Z    +0.000, E1  +361.710, E3 -389223.360}
SPL {X  -159.990, Y  +665.465, Z    +0.000, E1  +358.378, E3 -389224.277}
SPL {X  -159.990, Y  +661.791, Z    +0.000, E1  +355.213, E3 -389225.115}
SPL {X  -159.990, Y  +656.991, Z    +0.000, E1  +350.742, E3 -389226.534}
SPL {X  -159.990, Y  +648.067, Z    +0.000, E1  +342.328, E3 -389230.264}
SPL {X  -159.990, Y  +620.451, Z    +0.000, E1  +325.419, E3 -389254.111}
SPL {X  -159.990, Y  +591.256, Z    +0.000, E1  +319.966, E3 -389300.605}
SPL {X  -159.990, Y  +586.740, Z    +0.000, E1  +319.956, E3 -389311.995}
SPL {X  -159.990, Y  +581.814, Z    +0.000, E1  +319.956, E3 -389324.434}
SPL {X  -159.990, Y  +577.274, Z    +0.000, E1  +319.964, E3 -389335.912}
SPL {X  -159.990, Y  +572.933, Z    +0.000, E1  +319.959, E3 -389346.853}
SPL {X  -159.990, Y  +568.504, Z    +0.000, E1  +319.956, E3 -389358.016}
SPL {X  -159.990, Y  +564.427, Z    +0.000, E1  +319.959, E3 -389368.302}
SPL {X  -159.990, Y  +558.823, Z    +0.000, E1  +319.916, E3 -389382.381}
SPL {X  -159.990, Y  +553.571, Z    +0.000, E1  +319.954, E3 -389395.663}
SPL {X  -159.990, Y  +549.413, Z    +0.000, E1  +319.938, E3 -389406.129}
SPL {X  -159.990, Y  +544.924, Z    +0.000, E1  +319.955, E3 -389417.510}
SPL {X  -159.990, Y  +540.054, Z    +0.000, E1  +319.939, E3 -389429.796}
SPL {X  -159.990, Y  +535.835, Z    +0.000, E1  +319.966, E3 -389440.477}
SPL {X  -159.990, Y  +532.291, Z    +0.000, E1  +319.951, E3 -389449.385}
SPL {X  -159.990, Y  +527.393, Z    +0.000, E1  +319.924, E3 -389461.693}
SPL {X  -159.990, Y  +522.533, Z    +0.000, E1  +319.951, E3 -389473.991}
SPL {X  -159.990, Y  +496.806, Z    +0.000, E1  +312.216, E3 -389484.198}
SPL {X  -159.990, Y  +490.245, Z    +0.000, E1  +312.831, E3 -389500.730}
SPL {X  -159.990, Y  +486.737, Z    +0.000, E1  +313.729, E3 -389512.736}
SPL {X  -159.990, Y  +483.955, Z    +0.000, E1  +314.316, E3 -389522.028}
SPL {X  -159.990, Y  +480.580, Z    +0.000, E1  +315.242, E3 -389534.649}
SPL {X  -159.990, Y  +476.546, Z    +0.000, E1  +316.165, E3 -389548.944}
SPL {X  -159.990, Y  +473.377, Z    +0.000, E1  +316.953, E3 -389560.558}
SPL {X  -159.990, Y  +470.788, Z    +0.000, E1  +317.853, E3 -389571.972}
SPL {X  -159.990, Y  +467.944, Z    +0.000, E1  +318.635, E3 -389583.293}
SPL {X  -159.990, Y  +465.057, Z    +0.000, E1  +319.375, E3 -389594.858}
SPL {X  -159.990, Y  +461.409, Z    +0.000, E1  +319.848, E3 -389606.757}
SPL {X  -159.990, Y  +456.934, Z    +0.000, E1  +319.854, E3 -389618.033}
SPL {X  -159.990, Y  +452.940, Z    +0.000, E1  +319.854, E3 -389628.078}
SPL {X  -159.990, Y  +448.856, Z    +0.000, E1  +319.859, E3 -389638.361}
SPL {X  -159.990, Y  +443.741, Z    +0.000, E1  +319.827, E3 -389651.179}
SPL {X  -159.990, Y  +436.703, Z    +0.000, E1  +319.809, E3 -389668.861}
SPL {X  -159.990, Y  +430.690, Z    +0.000, E1  +319.854, E3 -389684.054}
SPL {X  -159.990, Y  +426.145, Z    +0.000, E1  +319.853, E3 -389695.494}
SPL {X  -159.990, Y  +421.880, Z    +0.000, E1  +319.860, E3 -389706.227}
SPL {X  -159.990, Y  +416.246, Z    +0.000, E1  +319.819, E3 -389720.355}
SPL {X  -159.990, Y  +409.936, Z    +0.000, E1  +319.849, E3 -389736.292}
SPL {X  -159.990, Y  +404.988, Z    +0.000, E1  +319.861, E3 -389748.758}
SPL {X  -159.990, Y  +400.535, Z    +0.000, E1  +319.859, E3 -389759.956}
SPL {X  -159.990, Y  +396.024, Z    +0.000, E1  +319.860, E3 -389771.312}
SPL {X  -159.990, Y  +391.614, Z    +0.000, E1  +319.860, E3 -389782.405}
SPL {X  -159.990, Y  +387.212, Z    +0.000, E1  +319.859, E3 -389793.478}
SPL {X  -159.990, Y  +382.743, Z    +0.000, E1  +319.857, E3 -389804.719}
SPL {X  -159.925, Y  +377.946, Z    +0.000, E1  +319.864, E3 -389816.856}
SPL {X  -159.703, Y  +372.915, Z    +0.000, E1  +319.904, E3 -389829.756}
SPL {X  -159.358, Y  +368.290, Z    +0.000, E1  +319.961, E3 -389841.718}
SPL {X  -158.955, Y  +364.333, Z    +0.000, E1  +320.046, E3 -389852.121}
SPL {X  -158.482, Y  +360.589, Z    +0.000, E1  +320.125, E3 -389862.047}
SPL {X  -157.729, Y  +355.695, Z    +0.000, E1  +320.237, E3 -389875.120}
SPL {X  -156.893, Y  +351.173, Z    +0.000, E1  +320.410, E3 -389887.403}
SPL {X  -156.148, Y  +347.650, Z    +0.000, E1  +320.549, E3 -389897.049}
SPL {X  -155.268, Y  +343.918, Z    +0.000, E1  +320.696, E3 -389907.330}
SPL {X  -154.153, Y  +339.677, Z    +0.000, E1  +320.896, E3 -389919.137}
SPL {X  -152.885, Y  +335.352, Z    +0.000, E1  +321.114, E3 -389931.291}
SPL {X  -151.010, Y  +329.654, Z    +0.000, E1  +326.674, E3 -389991.507}
ENDSPLINE

SPLINE
SPL {X  -157.513, Y  +354.453, Z    +0.000, E1  +340.941, E3 -390037.541}
SPL {X  -159.408, Y  +368.861, Z    +0.000, E1  +348.865, E3 -390046.964}
SPL {X  -159.941, Y  +378.532, Z    +0.000, E1  +354.551, E3 -390050.570}
SPL {X  -159.990, Y  +383.966, Z    +0.000, E1  +358.149, E3 -390052.021}
SPL {X  -159.990, Y  +388.001, Z    +0.000, E1  +361.086, E3 -390052.957}
SPL {X  -159.990, Y  +392.647, Z    +0.000, E1  +364.974, E3 -390054.095}
SPL {X  -159.990, Y  +397.943, Z    +0.000, E1  +369.963, E3 -390055.680}
SPL {X  -159.990, Y  +407.689, Z    +0.000, E1  +378.860, E3 -390060.334}
SPL {X  -159.990, Y  +434.822, Z    +0.000, E1  +394.625, E3 -390084.878}
SPL {X  -159.990, Y  +460.330, Z    +0.000, E1  +398.908, E3 -390129.154}
SPL {X  -159.990, Y  +464.953, Z    +0.000, E1  +398.907, E3 -390141.312}
SPL {X  -159.990, Y  +469.353, Z    +0.000, E1  +398.902, E3 -390152.892}
SPL {X  -159.990, Y  +475.034, Z    +0.000, E1  +398.936, E3 -390167.807}
SPL {X  -159.990, Y  +481.308, Z    +0.000, E1  +398.917, E3 -390184.318}
SPL {X  -159.990, Y  +485.396, Z    +0.000, E1  +398.893, E3 -390195.078}
SPL {X  -159.990, Y  +489.893, Z    +0.000, E1  +398.930, E3 -390206.833}
SPL {X  -159.990, Y  +496.271, Z    +0.000, E1  +398.942, E3 -390223.589}
SPL {X  -159.990, Y  +502.093, Z    +0.000, E1  +398.909, E3 -390238.973}
SPL {X  -159.990, Y  +506.629, Z    +0.000, E1  +398.900, E3 -390250.905}
SPL {X  -159.990, Y  +512.483, Z    +0.000, E1  +398.947, E3 -390266.234}
SPL {X  -159.990, Y  +518.435, Z    +0.000, E1  +398.905, E3 -390281.948}
SPL {X  -159.990, Y  +523.478, Z    +0.000, E1  +398.918, E3 -390295.176}
SPL {X  -159.990, Y  +528.627, Z    +0.000, E1  +398.910, E3 -390308.730}
SPL {X  -159.990, Y  +534.392, Z    +0.000, E1  +398.932, E3 -390323.860}
SPL {X  -159.990, Y  +540.299, Z    +0.000, E1  +398.912, E3 -390339.435}
SPL {X  -159.990, Y  +545.676, Z    +0.000, E1  +398.913, E3 -390353.572}
SPL {X  -159.990, Y  +550.777, Z    +0.000, E1  +398.906, E3 -390366.992}
SPL {X  -159.990, Y  +556.271, Z    +0.000, E1  +398.927, E3 -390381.394}
SPL {X  -159.990, Y  +561.696, Z    +0.000, E1  +398.912, E3 -390395.664}
SPL {X  -159.990, Y  +566.650, Z    +0.000, E1  +398.917, E3 -390408.677}
SPL {X  -159.990, Y  +571.814, Z    +0.000, E1  +398.914, E3 -390422.280}
SPL {X  -159.990, Y  +576.364, Z    +0.000, E1  +398.896, E3 -390434.283}
SPL {X  -159.990, Y  +582.060, Z    +0.000, E1  +398.942, E3 -390449.189}
SPL {X  -159.990, Y  +587.761, Z    +0.000, E1  +398.902, E3 -390464.238}
SPL {X  -159.990, Y  +592.962, Z    +0.000, E1  +398.925, E3 -390477.882}
SPL {X  -159.990, Y  +599.478, Z    +0.000, E1  +398.941, E3 -390494.992}
SPL {X  -159.990, Y  +606.904, Z    +0.000, E1  +398.953, E3 -390514.505}
SPL {X  -159.990, Y  +613.039, Z    +0.000, E1  +398.906, E3 -390530.705}
SPL {X  -159.990, Y  +618.087, Z    +0.000, E1  +398.915, E3 -390543.964}
SPL {X  -159.990, Y  +623.264, Z    +0.000, E1  +398.906, E3 -390557.598}
SPL {X  -159.990, Y  +628.669, Z    +0.000, E1  +398.928, E3 -390571.766}
SPL {X  -159.990, Y  +634.089, Z    +0.000, E1  +398.907, E3 -390586.042}
SPL {X  -159.990, Y  +638.639, Z    +0.000, E1  +398.904, E3 -390598.028}
SPL {X  -159.990, Y  +644.750, Z    +0.000, E1  +398.946, E3 -390614.033}
SPL {X  -159.990, Y  +650.458, Z    +0.000, E1  +398.900, E3 -390629.106}
SPL {X  -159.990, Y  +654.813, Z    +0.000, E1  +398.905, E3 -390640.550}
SPL {X  -159.990, Y  +660.353, Z    +0.000, E1  +398.930, E3 -390655.081}
SPL {X  -159.990, Y  +665.703, Z    +0.000, E1  +398.903, E3 -390669.189}
SPL {X  -159.990, Y  +671.472, Z    +0.000, E1  +398.942, E3 -390684.293}
SPL {X  -159.920, Y  +676.216, Z    +0.000, E1  +398.875, E3 -390696.928}
SPL {X  -159.761, Y  +680.061, Z    +0.000, E1  +398.873, E3 -390707.154}
SPL {X  -159.443, Y  +684.716, Z    +0.000, E1  +398.815, E3 -390719.719}
SPL {X  -158.962, Y  +689.604, Z    +0.000, E1  +398.740, E3 -390733.088}
SPL {X  -158.318, Y  +694.567, Z    +0.000, E1  +398.614, E3 -390746.849}
SPL {X  -157.472, Y  +699.775, Z    +0.000, E1  +398.483, E3 -390761.409}
SPL {X  -156.506, Y  +704.705, Z    +0.000, E1  +398.294, E3 -390775.409}
SPL {X  -155.680, Y  +708.387, Z    +0.000, E1  +398.127, E3 -390785.980}
SPL {X  -154.586, Y  +712.730, Z    +0.000, E1  +397.967, E3 -390798.477}
SPL {X  -153.345, Y  +717.131, Z    +0.000, E1  +397.713, E3 -390811.361}
SPL {X  -151.080, Y  +724.146, Z    +0.000, E1  +393.201, E3 -390869.815}
ENDSPLINE

SPLINE
SPL {X  -157.921, Y  +697.149, Z    +0.000, E1  +377.701, E3 -390921.376}
SPL {X  -159.579, Y  +682.959, Z    +0.000, E1  +369.793, E3 -390929.324}
SPL {X  -159.938, Y  +675.561, Z    +0.000, E1  +365.399, E3 -390931.746}
SPL {X  -159.990, Y  +669.910, Z    +0.000, E1  +361.710, E3 -390933.037}
SPL {X  -159.990, Y  +665.465, Z    +0.000, E1  +358.378, E3 -390933.955}
SPL {X  -159.990, Y  +661.791, Z    +0.000, E1  +355.213, E3 -390934.792}
SPL {X  -159.990, Y  +656.991, Z    +0.000, E1  +350.742, E3 -390936.212}
SPL {X  -159.990, Y  +648.067, Z    +0.000, E1  +342.328, E3 -390939.941}
SPL {X  -159.990, Y  +620.451, Z    +0.000, E1  +325.419, E3 -390963.789}
SPL {X  -159.990, Y  +591.256, Z    +0.000, E1  +319.966, E3 -391010.282}
SPL {X  -159.990, Y  +586.740, Z    +0.000, E1  +319.956, E3 -391021.672}
SPL {X  -159.990, Y  +581.814, Z    +0.000, E1  +319.956, E3 -391034.112}
SPL {X  -159.990, Y  +577.274, Z    +0.000, E1  +319.964, E3 -391045.589}
SPL {X  -159.990, Y  +572.933, Z    +0.000, E1  +319.959, E3 -391056.530}
SPL {X  -159.990, Y  +568.504, Z    +0.000, E1  +319.956, E3 -391067.693}
SPL {X  -159.990, Y  +564.427, Z    +0.000, E1  +319.959, E3 -391077.979}
SPL {X  -159.990, Y  +558.823, Z    +0.000, E1  +319.916, E3 -391092.059}
SPL {X  -159.990, Y  +553.571, Z    +0.000, E1  +319.954, E3 -391105.340}
SPL {X  -159.990, Y  +549.413, Z    +0.000, E1  +319.938, E3 -391115.806}
SPL {X  -159.990, Y  +543.439, Z    +0.000, E1  +319.921, E3 -391130.894}
SPL {X  -159.990, Y  +537.213, Z    +0.000, E1  +319.937, E3 -391146.637}
SPL {X  -159.990, Y  +530.667, Z    +0.000, E1  +319.910, E3 -391163.095}
SPL {X  -159.990, Y  +523.984, Z    +0.000, E1  +319.922, E3 -391179.961}
SPL {X  -159.990, Y  +496.806, Z    +0.000, E1  +312.216, E3 -391193.876}
SPL {X  -159.990, Y  +490.245, Z    +0.000, E1  +312.831, E3 -391210.407}
SPL {X  -159.990, Y  +484.831, Z    +0.000, E1  +314.066, E3 -391228.640}
SPL {X  -159.990, Y  +480.580, Z    +0.000, E1  +315.242, E3 -391244.326}
SPL {X  -159.990, Y  +476.546, Z    +0.000, E1  +316.165, E3 -391258.621}
SPL {X  -159.990, Y  +472.671, Z    +0.000, E1  +317.192, E3 -391273.448}
SPL {X  -159.990, Y  +468.809, Z    +0.000, E1  +318.343, E3 -391289.377}
SPL {X  -159.990, Y  +465.057, Z    +0.000, E1  +319.375, E3 -391304.535}
SPL {X  -159.990, Y  +461.409, Z    +0.000, E1  +319.848, E3 -391316.435}
SPL {X  -159.990, Y  +456.934, Z    +0.000, E1  +319.854, E3 -391327.710}
SPL {X  -159.990, Y  +452.940, Z    +0.000, E1  +319.854, E3 -391337.755}
SPL {X  -159.990, Y  +448.856, Z    +0.000, E1  +319.859, E3 -391348.038}
SPL {X  -159.990, Y  +443.741, Z    +0.000, E1  +319.827, E3 -391360.856}
SPL {X  -159.990, Y  +436.703, Z    +0.000, E1  +319.809, E3 -391378.538}
SPL {X  -159.990, Y  +430.690, Z    +0.000, E1  +319.854, E3 -391393.731}
SPL {X  -159.990, Y  +426.145, Z    +0.000, E1  +319.853, E3 -391405.171}
SPL {X  -159.990, Y  +421.880, Z    +0.000, E1  +319.860, E3 -391415.904}
SPL {X  -159.990, Y  +417.572, Z    +0.000, E1  +319.852, E3 -391426.731}
SPL {X  -159.990, Y  +412.619, Z    +0.000, E1  +319.850, E3 -391439.222}
SPL {X  -159.990, Y  +406.264, Z    +0.000, E1  +319.825, E3 -391455.170}
SPL {X  -159.990, Y  +400.535, Z    +0.000, E1  +319.859, E3 -391469.633}
SPL {X  -159.990, Y  +396.024, Z    +0.000, E1  +319.860, E3 -391480.989}
SPL {X  -159.990, Y  +391.614, Z    +0.000, E1  +319.860, E3 -391492.083}
SPL {X  -159.990, Y  +387.212, Z    +0.000, E1  +319.859, E3 -391503.155}
SPL {X  -159.990, Y  +382.743, Z    +0.000, E1  +319.857, E3 -391514.396}
SPL {X  -159.925, Y  +377.946, Z    +0.000, E1  +319.864, E3 -391526.533}
SPL {X  -159.703, Y  +372.915, Z    +0.000, E1  +319.904, E3 -391539.433}
SPL {X  -159.358, Y  +368.290, Z    +0.000, E1  +319.961, E3 -391551.396}
SPL {X  -158.955, Y  +364.333, Z    +0.000, E1  +320.046, E3 -391561.798}
SPL {X  -158.482, Y  +360.589, Z    +0.000, E1  +320.125, E3 -391571.725}
SPL {X  -157.729, Y  +355.695, Z    +0.000, E1  +320.237, E3 -391584.797}
SPL {X  -156.893, Y  +351.173, Z    +0.000, E1  +320.410, E3 -391597.080}
SPL {X  -156.148, Y  +347.650, Z    +0.000, E1  +320.549, E3 -391606.726}
SPL {X  -155.268, Y  +343.918, Z    +0.000, E1  +320.696, E3 -391617.007}
SPL {X  -153.936, Y  +338.906, Z    +0.000, E1  +320.911, E3 -391630.946}
SPL {X  -152.628, Y  +334.526, Z    +0.000, E1  +321.188, E3 -391643.348}
SPL {X  -151.010, Y  +329.654, Z    +0.000, E1  +326.674, E3 -391701.184}
ENDSPLINE

SPLINE
SPL {X  -157.513, Y  +354.453, Z    +0.000, E1  +340.941, E3 -391747.219}
SPL {X  -159.408, Y  +368.861, Z    +0.000, E1  +348.865, E3 -391756.641}
SPL {X  -159.941, Y  +378.532, Z    +0.000, E1  +354.551, E3 -391760.247}
SPL {X  -159.990, Y  +383.966, Z    +0.000, E1  +358.149, E3 -391761.699}
SPL {X  -159.990, Y  +388.001, Z    +0.000, E1  +361.086, E3 -391762.634}
SPL {X  -159.990, Y  +392.647, Z    +0.000, E1  +364.974, E3 -391763.773}
SPL {X  -159.990, Y  +397.943, Z    +0.000, E1  +369.963, E3 -391765.357}
SPL {X  -159.990, Y  +407.689, Z    +0.000, E1  +378.860, E3 -391770.012}
SPL {X  -159.990, Y  +434.822, Z    +0.000, E1  +394.625, E3 -391794.556}
SPL {X  -159.990, Y  +460.330, Z    +0.000, E1  +398.908, E3 -391838.831}
SPL {X  -159.990, Y  +464.953, Z    +0.000, E1  +398.907, E3 -391850.989}
SPL {X  -159.990, Y  +469.353, Z    +0.000, E1  +398.902, E3 -391862.570}
SPL {X  -159.990, Y  +475.034, Z    +0.000, E1  +398.936, E3 -391877.485}
SPL {X  -159.990, Y  +481.308, Z    +0.000, E1  +398.917, E3 -391893.995}
SPL {X  -159.990, Y  +485.396, Z    +0.000, E1  +398.893, E3 -391904.755}
SPL {X  -159.990, Y  +489.893, Z    +0.000, E1  +398.930, E3 -391916.510}
SPL {X  -159.990, Y  +496.271, Z    +0.000, E1  +398.942, E3 -391933.267}
SPL {X  -159.990, Y  +502.093, Z    +0.000, E1  +398.909, E3 -391948.651}
SPL {X  -159.990, Y  +507.821, Z    +0.000, E1  +398.930, E3 -391963.671}
SPL {X  -159.990, Y  +513.533, Z    +0.000, E1  +398.910, E3 -391978.730}
SPL {X  -159.990, Y  +518.435, Z    +0.000, E1  +398.905, E3 -391991.625}
SPL {X  -159.990, Y  +523.478, Z    +0.000, E1  +398.918, E3 -392004.854}
SPL {X  -159.990, Y  +528.627, Z    +0.000, E1  +398.910, E3 -392018.407}
SPL {X  -159.990, Y  +533.053, Z    +0.000, E1  +398.899, E3 -392030.065}
SPL {X  -159.990, Y  +537.174, Z    +0.000, E1  +398.910, E3 -392040.879}
SPL {X  -159.990, Y  +541.259, Z    +0.000, E1  +398.888, E3 -392051.679}
SPL {X  -159.990, Y  +545.676, Z    +0.000, E1  +398.913, E3 -392063.250}
SPL {X  -159.990, Y  +550.777, Z    +0.000, E1  +398.906, E3 -392076.669}
SPL {X  -159.990, Y  +554.638, Z    +0.000, E1  +398.890, E3 -392086.840}
SPL {X  -159.990, Y  +557.678, Z    +0.000, E1  +398.893, E3 -392094.816}
SPL {X  -159.990, Y  +561.696, Z    +0.000, E1  +398.912, E3 -392105.341}
SPL {X  -159.990, Y  +566.650, Z    +0.000, E1  +398.917, E3 -392118.355}
SPL {X  -159.990, Y  +571.814, Z    +0.000, E1  +398.914, E3 -392131.957}
SPL {X  -159.990, Y  +576.364, Z    +0.000, E1  +398.896, E3 -392143.961}
SPL {X  -159.990, Y  +582.060, Z    +0.000, E1  +398.942, E3 -392158.866}
SPL {X  -159.990, Y  +589.106, Z    +0.000, E1  +398.939, E3 -392177.398}
SPL {X  -159.990, Y  +596.185, Z    +0.000, E1  +398.945, E3 -392196.006}
SPL {X  -159.990, Y  +602.727, Z    +0.000, E1  +398.920, E3 -392213.246}
SPL {X  -159.990, Y  +608.112, Z    +0.000, E1  +398.911, E3 -392227.420}
SPL {X  -159.990, Y  +614.125, Z    +0.000, E1  +398.936, E3 -392243.195}
SPL {X  -159.990, Y  +619.061, Z    +0.000, E1  +398.894, E3 -392256.227}
SPL {X  -159.990, Y  +623.264, Z    +0.000, E1  +398.906, E3 -392267.276}
SPL {X  -159.990, Y  +628.669, Z    +0.000, E1  +398.928, E3 -392281.444}
SPL {X  -159.990, Y  +634.089, Z    +0.000, E1  +398.907, E3 -392295.720}
SPL {X  -159.990, Y  +638.639, Z    +0.000, E1  +398.904, E3 -392307.705}
SPL {X  -159.990, Y  +644.750, Z    +0.000, E1  +398.946, E3 -392323.711}
SPL {X  -159.990, Y  +650.458, Z    +0.000, E1  +398.900, E3 -392338.783}
SPL {X  -159.990, Y  +654.813, Z    +0.000, E1  +398.905, E3 -392350.227}
SPL {X  -159.990, Y  +660.353, Z    +0.000, E1  +398.930, E3 -392364.759}
SPL {X  -159.990, Y  +665.703, Z    +0.000, E1  +398.903, E3 -392378.866}
SPL {X  -159.990, Y  +669.966, Z    +0.000, E1  +398.902, E3 -392390.073}
SPL {X  -159.954, Y  +674.895, Z    +0.000, E1  +398.910, E3 -392403.052}
SPL {X  -159.761, Y  +680.061, Z    +0.000, E1  +398.873, E3 -392416.831}
SPL {X  -159.327, Y  +686.045, Z    +0.000, E1  +398.835, E3 -392432.954}
SPL {X  -158.832, Y  +690.714, Z    +0.000, E1  +398.685, E3 -392445.880}
SPL {X  -158.318, Y  +694.567, Z    +0.000, E1  +398.614, E3 -392456.527}
SPL {X  -157.472, Y  +699.775, Z    +0.000, E1  +398.483, E3 -392471.087}
SPL {X  -156.506, Y  +704.705, Z    +0.000, E1  +398.294, E3 -392485.087}
SPL {X  -155.357, Y  +709.721, Z    +0.000, E1  +398.108, E3 -392499.442}
SPL {X  -154.286, Y  +713.838, Z    +0.000, E1  +397.877, E3 -392511.425}
SPL {X  -153.345, Y  +717.131, Z    +0.000, E1  +397.713, E3 -392521.039}
SPL {X  -151.080, Y  +724.146, Z    +0.000, E1  +393.201, E3 -392579.493}
ENDSPLINE

SPLINE
SPL {X  -157.921, Y  +697.149, Z    +0.000, E1  +377.701, E3 -392631.053}
SPL {X  -159.579, Y  +682.959, Z    +0.000, E1  +369.793, E3 -392639.002}
SPL {X  -159.938, Y  +675.561, Z    +0.000, E1  +365.399, E3 -392641.424}
SPL {X  -159.990, Y  +669.910, Z    +0.000, E1  +361.710, E3 -392642.715}
SPL {X  -159.990, Y  +665.465, Z    +0.000, E1  +358.378, E3 -392643.632}
SPL {X  -159.990, Y  +661.791, Z    +0.000, E1  +355.213, E3 -392644.470}
SPL {X  -159.990, Y  +656.991, Z    +0.000, E1  +350.742, E3 -392645.889}
SPL {X  -159.990, Y  +649.722, Z    +0.000, E1  +343.777, E3 -392648.808}
SPL {X  -159.990, Y  +645.752, Z    +0.000, E1  +340.157, E3 -392650.749}
SPL {X  -159.990, Y  +620.451, Z    +0.000, E1  +325.419, E3 -392673.466}
SPL {X  -159.990, Y  +591.256, Z    +0.000, E1  +319.966, E3 -392719.959}
SPL {X  -159.990, Y  +586.740, Z    +0.000, E1  +319.956, E3 -392731.350}
SPL {X  -159.990, Y  +581.814, Z    +0.000, E1  +319.956, E3 -392743.789}
SPL {X  -159.990, Y  +577.274, Z    +0.000, E1  +319.964, E3 -392755.267}
SPL {X  -159.990, Y  +572.933, Z    +0.000, E1  +319.959, E3 -392766.208}
SPL {X  -159.990, Y  +568.504, Z    +0.000, E1  +319.956, E3 -392777.371}
SPL {X  -159.990, Y  +563.189, Z    +0.000, E1  +319.932, E3 -392790.744}
SPL {X  -159.990, Y  +557.707, Z    +0.000, E1  +319.949, E3 -392804.599}
SPL {X  -159.990, Y  +553.571, Z    +0.000, E1  +319.954, E3 -392815.018}
SPL {X  -159.990, Y  +549.413, Z    +0.000, E1  +319.938, E3 -392825.484}
SPL {X  -159.990, Y  +544.924, Z    +0.000, E1  +319.955, E3 -392836.865}
SPL {X  -159.990, Y  +540.054, Z    +0.000, E1  +319.939, E3 -392849.151}
SPL {X  -159.990, Y  +535.835, Z    +0.000, E1  +319.966, E3 -392859.831}
SPL {X  -159.990, Y  +532.291, Z    +0.000, E1  +319.951, E3 -392868.740}
SPL {X  -159.990, Y  +527.393, Z    +0.000, E1  +319.924, E3 -392881.048}
SPL {X  -159.990, Y  +522.533, Z    +0.000, E1  +319.951, E3 -392893.346}
SPL {X  -159.990, Y  +502.378, Z    +0.000, E1  +313.079, E3 -392897.750}
SPL {X  -159.990, Y  +493.568, Z    +0.000, E1  +312.053, E3 -392908.917}
SPL {X  -159.990, Y  +489.464, Z    +0.000, E1  +313.059, E3 -392922.784}
SPL {X  -159.990, Y  +484.831, Z    +0.000, E1  +314.066, E3 -392938.317}
SPL {X  -159.990, Y  +480.580, Z    +0.000, E1  +315.242, E3 -392954.004}
SPL {X  -159.990, Y  +476.546, Z    +0.000, E1  +316.165, E3 -392968.298}
SPL {X  -159.990, Y  +473.377, Z    +0.000, E1  +316.953, E3 -392979.913}
SPL {X  -159.990, Y  +470.788, Z    +0.000, E1  +317.853, E3 -392991.326}
SPL {X  -159.990, Y  +467.944, Z    +0.000, E1  +318.635, E3 -393002.647}
SPL {X  -159.990, Y  +465.057, Z    +0.000, E1  +319.375, E3 -393014.213}
SPL {X  -159.990, Y  +461.409, Z    +0.000, E1  +319.848, E3 -393026.112}
SPL {X  -159.990, Y  +456.934, Z    +0.000, E1  +319.854, E3 -393037.388}
SPL {X  -159.990, Y  +452.940, Z    +0.000, E1  +319.854, E3 -393047.432}
SPL {X  -159.990, Y  +448.856, Z    +0.000, E1  +319.859, E3 -393057.716}
SPL {X  -159.990, Y  +444.973, Z    +0.000, E1  +319.856, E3 -393067.481}
SPL {X  -159.990, Y  +439.927, Z    +0.000, E1  +319.837, E3 -393080.138}
SPL {X  -159.990, Y  +435.246, Z    +0.000, E1  +319.853, E3 -393091.947}
SPL {X  -159.990, Y  +430.690, Z    +0.000, E1  +319.854, E3 -393103.409}
SPL {X  -159.990, Y  +426.145, Z    +0.000, E1  +319.853, E3 -393114.848}
SPL {X  -159.990, Y  +421.880, Z    +0.000, E1  +319.860, E3 -393125.581}
SPL {X  -159.990, Y  +417.572, Z    +0.000, E1  +319.852, E3 -393136.408}
SPL {X  -159.990, Y  +412.619, Z    +0.000, E1  +319.850, E3 -393148.900}
SPL {X  -159.990, Y  +406.264, Z    +0.000, E1  +319.825, E3 -393164.848}
SPL {X  -159.990, Y  +400.535, Z    +0.000, E1  +319.859, E3 -393179.311}
SPL {X  -159.990, Y  +396.024, Z    +0.000, E1  +319.860, E3 -393190.667}
SPL {X  -159.990, Y  +391.614, Z    +0.000, E1  +319.860, E3 -393201.760}
SPL {X  -159.990, Y  +387.212, Z    +0.000, E1  +319.859, E3 -393212.832}
SPL {X  -159.990, Y  +382.743, Z    +0.000, E1  +319.857, E3 -393224.074}
SPL {X  -159.925, Y  +377.946, Z    +0.000, E1  +319.864, E3 -393236.211}
SPL {X  -159.703, Y  +372.915, Z    +0.000, E1  +319.904, E3 -393249.111}
SPL {X  -159.358, Y  +368.290, Z    +0.000, E1  +319.961, E3 -393261.073}
SPL {X  -158.955, Y  +364.333, Z    +0.000, E1  +320.046, E3 -393271.476}
SPL {X  -158.270, Y  +359.106, Z    +0.000, E1  +320.118, E3 -393285.287}
SPL {X  -157.143, Y  +352.453, Z    +0.000, E1  +320.322, E3 -393303.217}
SPL {X  -156.148, Y  +347.650, Z    +0.000, E1  +320.549, E3 -393316.404}
SPL {X  -155.268, Y  +343.918, Z    +0.000, E1  +320.696, E3 -393326.685}
SPL {X  -154.153, Y  +339.677, Z    +0.000, E1  +320.896, E3 -393338.491}
SPL {X  -152.885, Y  +335.352, Z    +0.000, E1  +321.114, E3 -393350.646}
SPL {X  -151.010, Y  +329.654, Z    +0.000, E1  +326.674, E3 -393410.862}
ENDSPLINE

SPLINE
SPL {X  -157.513, Y  +354.453, Z    +0.000, E1  +340.941, E3 -393456.896}
SPL {X  -159.638, Y  +371.886, Z    +0.000, E1  +350.545, E3 -393467.558}
SPL {X  -159.990, Y  +382.357, Z    +0.000, E1  +356.972, E3 -393470.973}
SPL {X  -159.990, Y  +388.001, Z    +0.000, E1  +361.086, E3 -393472.311}
SPL {X  -159.990, Y  +392.647, Z    +0.000, E1  +364.974, E3 -393473.450}
SPL {X  -159.990, Y  +397.943, Z    +0.000, E1  +369.963, E3 -393475.035}
SPL {X  -159.990, Y  +407.689, Z    +0.000, E1  +378.860, E3 -393479.689}
SPL {X  -159.990, Y  +434.822, Z    +0.000, E1  +394.625, E3 -393504.233}
SPL {X  -159.990, Y  +460.330, Z    +0.000, E1  +398.908, E3 -393548.509}
SPL {X  -159.990, Y  +464.953, Z    +0.000, E1  +398.907, E3 -393560.667}
SPL {X  -159.990, Y  +469.353, Z    +0.000, E1  +398.902, E3 -393572.247}
SPL {X  -159.990, Y  +475.034, Z    +0.000, E1  +398.936, E3 -393587.162}
SPL {X  -159.990, Y  +481.308, Z    +0.000, E1  +398.917, E3 -393603.673}
SPL {X  -159.990, Y  +485.396, Z    +0.000, E1  +398.893, E3 -393614.432}
SPL {X  -159.990, Y  +489.893, Z    +0.000, E1  +398.930, E3 -393626.188}
SPL {X  -159.990, Y  +496.271, Z    +0.000, E1  +398.942, E3 -393642.944}
SPL {X  -159.990, Y  +502.093, Z    +0.000, E1  +398.909, E3 -393658.328}
SPL {X  -159.990, Y  +506.629, Z    +0.000, E1  +398.900, E3 -393670.260}
SPL {X  -159.990, Y  +512.483, Z    +0.000, E1  +398.947, E3 -393685.589}
SPL {X  -159.990, Y  +518.435, Z    +0.000, E1  +398.905, E3 -393701.303}
SPL {X  -159.990, Y  +523.478, Z    +0.000, E1  +398.918, E3 -393714.531}
SPL {X  -159.990, Y  +528.627, Z    +0.000, E1  +398.910, E3 -393728.085}
SPL {X  -159.990, Y  +534.392, Z    +0.000, E1  +398.932, E3 -393743.215}
SPL {X  -159.990, Y  +540.299, Z    +0.000, E1  +398.912, E3 -393758.790}
SPL {X  -159.990, Y  +545.676, Z    +0.000, E1  +398.913, E3 -393772.927}
SPL {X  -159.990, Y  +550.777, Z    +0.000, E1  +398.906, E3 -393786.346}
SPL {X  -159.990, Y  +556.271, Z    +0.000, E1  +398.927, E3 -393800.749}
SPL {X  -159.990, Y  +561.696, Z    +0.000, E1  +398.912, E3 -393815.018}
SPL {X  -159.990, Y  +566.650, Z    +0.000, E1  +398.917, E3 -393828.032}
SPL {X  -159.990, Y  +571.814, Z    +0.000, E1  +398.914, E3 -393841.635}
SPL {X  -159.990, Y  +576.364, Z    +0.000, E1  +398.896, E3 -393853.638}
SPL {X  -159.990, Y  +582.060, Z    +0.000, E1  +398.942, E3 -393868.544}
SPL {X  -159.990, Y  +587.761, Z    +0.000, E1  +398.902, E3 -393883.593}
SPL {X  -159.990, Y  +592.962, Z    +0.000, E1  +398.925, E3 -393897.237}
SPL {X  -159.990, Y  +599.478, Z    +0.000, E1  +398.941, E3 -393914.347}
SPL {X  -159.990, Y  +606.904, Z    +0.000, E1  +398.953, E3 -393933.860}
SPL {X  -159.990, Y  +613.039, Z    +0.000, E1  +398.906, E3 -393950.060}
SPL {X  -159.990, Y  +618.087, Z    +0.000, E1  +398.915, E3 -393963.319}
SPL {X  -159.990, Y  +623.264, Z    +0.000, E1  +398.906, E3 -393976.953}
SPL {X  -159.990, Y  +628.669, Z    +0.000, E1  +398.928, E3 -393991.121}
SPL {X  -159.990, Y  +634.089, Z    +0.000, E1  +398.907, E3 -394005.397}
SPL {X  -159.990, Y  +638.639, Z    +0.000, E1  +398.904, E3 -394017.383}
SPL {X  -159.990, Y  +644.750, Z    +0.000, E1  +398.946, E3 -394033.388}
SPL {X  -159.990, Y  +650.458, Z    +0.000, E1  +398.900, E3 -394048.460}
SPL {X  -159.990, Y  +654.813, Z    +0.000, E1  +398.905, E3 -394059.905}
SPL {X  -159.990, Y  +660.353, Z    +0.000, E1  +398.930, E3 -394074.436}
SPL {X  -159.990, Y  +665.703, Z    +0.000, E1  +398.903, E3 -394088.543}
SPL {X  -159.990, Y  +671.472, Z    +0.000, E1  +398.942, E3 -394103.648}
SPL {X  -159.920, Y  +676.216, Z    +0.000, E1  +398.875, E3 -394116.283}
SPL {X  -159.761, Y  +680.061, Z    +0.000, E1  +398.873, E3 -394126.509}
SPL {X  -159.443, Y  +684.716, Z    +0.000, E1  +398.815, E3 -394139.074}
SPL {X  -158.962, Y  +689.604, Z    +0.000, E1  +398.740, E3 -394152.443}
SPL {X  -158.318, Y  +694.567, Z    +0.000, E1  +398.614, E3 -394166.204}
SPL {X  -157.472, Y  +699.775, Z    +0.000, E1  +398.483, E3 -394180.764}
SPL {X  -156.506, Y  +704.705, Z    +0.000, E1  +398.294, E3 -394194.764}
SPL {X  -155.680, Y  +708.387, Z    +0.000, E1  +398.127, E3 -394205.335}
SPL {X  -154.586, Y  +712.730, Z    +0.000, E1  +397.967, E3 -394217.832}
SPL {X  -153.345, Y  +717.131, Z    +0.000, E1  +397.713, E3 -394230.716}
SPL {X  -151.080, Y  +724.146, Z    +0.000, E1  +393.201, E3 -394289.170}
ENDSPLINE

SPLINE
SPL {X  -157.921, Y  +697.149, Z    +0.000, E1  +377.701, E3 -394340.731}
SPL {X  -159.579, Y  +682.959, Z    +0.000, E1  +369.793, E3 -394348.679}
SPL {X  -159.938, Y  +675.561, Z    +0.000, E1  +365.399, E3 -394351.101}
SPL {X  -159.990, Y  +669.910, Z    +0.000, E1  +361.710, E3 -394352.392}
SPL {X  -159.990, Y  +665.465, Z    +0.000, E1  +358.378, E3 -394353.310}
SPL {X  -159.990, Y  +661.791, Z    +0.000, E1  +355.213, E3 -394354.147}
SPL {X  -159.990, Y  +656.991, Z    +0.000, E1  +350.742, E3 -394355.567}
SPL {X  -159.990, Y  +648.067, Z    +0.000, E1  +342.328, E3 -394359.296}
SPL {X  -159.990, Y  +620.451, Z    +0.000, E1  +325.419, E3 -394383.143}
SPL {X  -159.990, Y  +591.256, Z    +0.000, E1  +319.966, E3 -394429.637}
SPL {X  -159.990, Y  +586.740, Z    +0.000, E1  +319.956, E3 -394441.027}
SPL {X  -159.990, Y  +581.814, Z    +0.000, E1  +319.956, E3 -394453.467}
SPL {X  -159.990, Y  +577.274, Z    +0.000, E1  +319.964, E3 -394464.944}
SPL {X  -159.990, Y  +572.933, Z    +0.000, E1  +319.959, E3 -394475.885}
SPL {X  -159.990, Y  +568.504, Z    +0.000, E1  +319.956, E3 -394487.048}
SPL {X  -159.990, Y  +563.189, Z    +0.000, E1  +319.932, E3 -394500.421}
SPL {X  -159.990, Y  +557.707, Z    +0.000, E1  +319.949, E3 -394514.277}
SPL {X  -159.990, Y  +552.104, Z    +0.000, E1  +319.922, E3 -394528.352}
SPL {X  -159.990, Y  +545.912, Z    +0.000, E1  +319.929, E3 -394544.001}
SPL {X  -159.990, Y  +540.054, Z    +0.000, E1  +319.939, E3 -394558.828}
SPL {X  -159.990, Y  +533.683, Z    +0.000, E1  +319.916, E3 -394574.853}
SPL {X  -159.990, Y  +527.393, Z    +0.000, E1  +319.924, E3 -394590.726}
SPL {X  -159.990, Y  +522.533, Z    +0.000, E1  +319.951, E3 -394603.023}
SPL {X  -159.990, Y  +502.378, Z    +0.000, E1  +313.079, E3 -394607.427}
SPL {X  -159.990, Y  +493.568, Z    +0.000, E1  +312.053, E3 -394618.595}
SPL {X  -159.990, Y  +489.464, Z    +0.000, E1  +313.059, E3 -394632.461}
SPL {X  -159.990, Y  +484.831, Z    +0.000, E1  +314.066, E3 -394647.995}
SPL {X  -159.990, Y  +480.580, Z    +0.000, E1  +315.242, E3 -394663.681}
SPL {X  -159.990, Y  +476.546, Z    +0.000, E1  +316.165, E3 -394677.976}
SPL {X  -159.990, Y  +472.671, Z    +0.000, E1  +317.192, E3 -394692.803}
SPL {X  -159.990, Y  +468.809, Z    +0.000, E1  +318.343, E3 -394708.732}
SPL {X  -159.990, Y  +465.057, Z    +0.000, E1  +319.375, E3 -394723.890}
ENDSPLINE

SPLINE
SPL {X  -159.990, Y  +491.634, Z    +0.000, E1  +334.596, E3 -394736.681}
ENDSPLINE

